KUKA KRL program: MyProgram_018().src

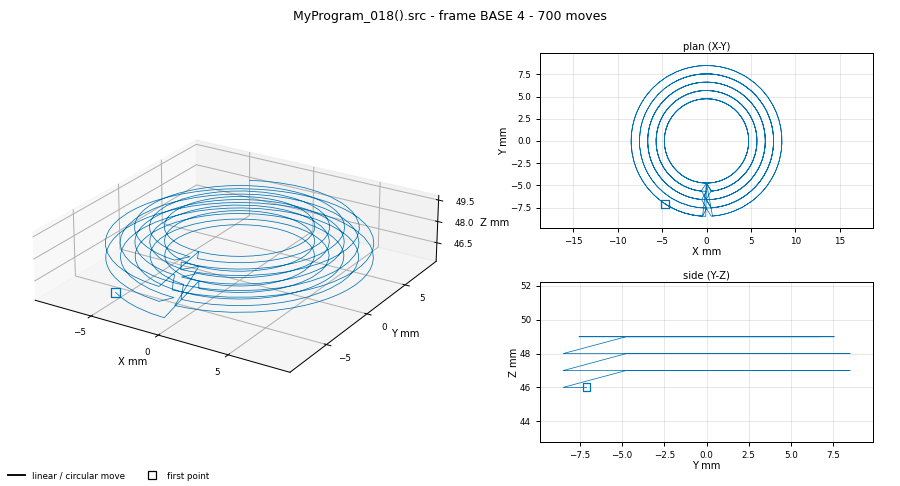
[picture p0: tool path of MyProgram_018().src in frame BASE 4, 700 of 700 moves have a stored position in this frame; points joined in program order, loops and branches not executed]
&ACCESS RVP
&REL 1
&PARAM TEMPLATE = C:\KRC\Roboter\Template\vorgabe
&PARAM EDITMASK = *
DEF MyProgram_018()
; ---- Setting reference (Base) ----
$BASE = BASE_DATA[4]

; --------------------------
; ---- Setting tool (TCP) ----
$TOOL = TOOL_DATA[3]
; --------------------------

$VEL.CP = VEL_APROX_PRINT
Startdeposition()
$VEL.CP = VEL_PRINT
LIN {X -4.657,Y -7.0952,Z 46,A -3.1359,B 0,C 0,E1 0.1598,E2 90.0712} C_DIS
LIN {X -3.9154,Y -7.53,Z 46,A -3.1272,B 0,C 0,E1 0.1598,E2 90.0712} C_DIS
LIN {X -3.1336,Y -7.8876,Z 46,A -3.1138,B 0,C 0,E1 0.1598,E2 90.0713} C_DIS
LIN {X -2.3197,Y -8.1643,Z 46,A -3.0957,B 0,C 0,E1 0.1598,E2 90.0714} C_DIS
LIN {X -1.1138,Y -8.4186,Z 46,A -3.0624,B 0,C 0,E1 0.1598,E2 90.0714} C_DIS
LIN {X -0.0867,Y -8.4896,Z 46,A -3.0278,B 0,C 0,E1 0.1598,E2 90.0715} C_DIS
Enddeposition()
LIN {X 0.0009,Y -4.7549,Z 47,A -2.851,B 0,C 0,E1 0.1598,E2 90.0604} C_DIS
Startdeposition()
$VEL.CP = VEL_PRINT
LIN {X 0.0009,Y -4.7549,Z 47,A -2.8568,B 0,C 0,E1 0.1598,E2 90.0661} C_DIS
LIN {X -0.8332,Y -4.6769,Z 47,A -2.889,B 0,C 0,E1 0.1598,E2 90.071} C_DIS
LIN {X -1.4834,Y -4.5141,Z 47,A -2.9065,B 0,C 0,E1 0.1598,E2 90.0716} C_DIS
LIN {X -2.1038,Y -4.2602,Z 47,A -2.9185,B 0,C 0,E1 0.1598,E2 90.0716} C_DIS
LIN {X -2.6818,Y -3.9209,Z 47,A -2.9253,B 0,C 0,E1 0.1598,E2 90.0716} C_DIS
LIN {X -3.2068,Y -3.5044,Z 47,A -2.9268,B 0,C 0,E1 0.1598,E2 90.0716} C_DIS
LIN {X -3.668,Y -3.0182,Z 47,A -2.9231,B 0,C 0,E1 0.1598,E2 90.0716} C_DIS
LIN {X -4.0561,Y -2.4717,Z 47,A -2.9141,B 0,C 0,E1 0.1598,E2 90.0716} C_DIS
LIN {X -4.3653,Y -1.8772,Z 47,A -2.9002,B 0,C 0,E1 0.1598,E2 90.0716} C_DIS
LIN {X -4.5856,Y -1.244,Z 47,A -2.8814,B 0,C 0,E1 0.1598,E2 90.0716} C_DIS
LIN {X -4.7134,Y -0.5861,Z 47,A -2.8582,B 0,C 0,E1 0.1598,E2 90.0716} C_DIS
LIN {X -4.7503,Y 0.0831,Z 47,A -2.8312,B 0,C 0,E1 0.1598,E2 90.0716} C_DIS
LIN {X -4.6907,Y 0.7507,Z 47,A -2.8007,B 0,C 0,E1 0.1598,E2 90.0716} C_DIS
LIN {X -4.5372,Y 1.4029,Z 47,A -2.7674,B 0,C 0,E1 0.1598,E2 90.0716} C_DIS
LIN {X -4.2974,Y 2.0289,Z 47,A -2.732,B 0,C 0,E1 0.1598,E2 90.0717} C_DIS
LIN {X -3.9689,Y 2.6132,Z 47,A -2.6952,B 0,C 0,E1 0.1598,E2 90.0718} C_DIS
LIN {X -3.5614,Y 3.1455,Z 47,A -2.6576,B 0,C 0,E1 0.1598,E2 90.0718} C_DIS
LIN {X -3.0827,Y 3.6147,Z 47,A -2.6201,B 0,C 0,E1 0.1598,E2 90.072} C_DIS
LIN {X -2.5433,Y 4.0125,Z 47,A -2.5834,B 0,C 0,E1 0.1598,E2 90.072} C_DIS
LIN {X -1.8762,Y 4.3636,Z 47,A -2.5439,B 0,C 0,E1 0.1598,E2 90.0721} C_DIS
LIN {X -1.3241,Y 4.5617,Z 47,A -2.5152,B 0,C 0,E1 0.1598,E2 90.0721} C_DIS
LIN {X -0.6691,Y 4.7028,Z 47,A -2.4851,B 0,C 0,E1 0.1598,E2 90.0722} C_DIS
LIN {X -0.0005,Y 4.7507,Z 47,A -2.4584,B 0,C 0,E1 0.1598,E2 90.0722} C_DIS
LIN {X 0.6681,Y 4.7041,Z 47,A -2.4358,B 0,C 0,E1 0.1598,E2 90.0723} C_DIS
LIN {X 1.3234,Y 4.5632,Z 47,A -2.4176,B 0,C 0,E1 0.1598,E2 90.0723} C_DIS
LIN {X 1.9524,Y 4.3316,Z 47,A -2.4042,B 0,C 0,E1 0.1598,E2 90.0723} C_DIS
LIN {X 2.5429,Y 4.0145,Z 47,A -2.3959,B 0,C 0,E1 0.1598,E2 90.0723} C_DIS
LIN {X 3.0827,Y 3.6169,Z 47,A -2.3929,B 0,C 0,E1 0.1598,E2 90.0723} C_DIS
LIN {X 3.5609,Y 3.147,Z 47,A -2.3953,B 0,C 0,E1 0.1598,E2 90.0723} C_DIS
LIN {X 3.9682,Y 2.6145,Z 47,A -2.4029,B 0,C 0,E1 0.1598,E2 90.0722} C_DIS
LIN {X 4.2968,Y 2.0301,Z 47,A -2.4157,B 0,C 0,E1 0.1598,E2 90.0722} C_DIS
LIN {X 4.5388,Y 1.4049,Z 47,A -2.4334,B 0,C 0,E1 0.1598,E2 90.0721} C_DIS
LIN {X 4.6912,Y 0.7522,Z 47,A -2.4556,B 0,C 0,E1 0.1598,E2 90.0721} C_DIS
LIN {X 4.7506,Y 0.0846,Z 47,A -2.4818,B 0,C 0,E1 0.1598,E2 90.0721} C_DIS
LIN {X 4.7139,Y -0.5846,Z 47,A -2.5117,B 0,C 0,E1 0.1598,E2 90.072} C_DIS
LIN {X 4.5853,Y -1.2422,Z 47,A -2.5445,B 0,C 0,E1 0.1598,E2 90.072} C_DIS
LIN {X 4.3647,Y -1.875,Z 47,A -2.5796,B 0,C 0,E1 0.1598,E2 90.072} C_DIS
LIN {X 4.0578,Y -2.4707,Z 47,A -2.6163,B 0,C 0,E1 0.1598,E2 90.0719} C_DIS
LIN {X 3.6688,Y -3.0165,Z 47,A -2.6539,B 0,C 0,E1 0.1598,E2 90.0719} C_DIS
LIN {X 3.2079,Y -3.5028,Z 47,A -2.6916,B 0,C 0,E1 0.1598,E2 90.0719} C_DIS
LIN {X 2.6838,Y -3.9208,Z 47,A -2.7287,B 0,C 0,E1 0.1598,E2 90.0719} C_DIS
LIN {X 2.1055,Y -4.2599,Z 47,A -2.7644,B 0,C 0,E1 0.1598,E2 90.0719} C_DIS
LIN {X 1.4853,Y -4.5146,Z 47,A -2.798,B 0,C 0,E1 0.1598,E2 90.0719} C_DIS
LIN {X 0.8353,Y -4.6792,Z 47,A -2.8289,B 0,C 0,E1 0.1598,E2 90.0718} C_DIS
LIN {X 0.0009,Y -4.7549,Z 47,A -2.8628,B 0,C 0,E1 0.1598,E2 90.0718} C_DIS
Enddeposition()
LIN {X 0.0009,Y -4.7549,Z 47,A -2.8628,B 0,C 0,E1 0.1598,E2 90.0718} C_DIS
Startdeposition()
$VEL.CP = VEL_PRINT
LIN {X 0.5845,Y -5.6535,Z 47,A -2.8792,B 0,C 0,E1 0.1598,E2 90.0712} C_DIS
LIN {X 1.3635,Y -5.516,Z 47,A -2.8453,B 0,C 0,E1 0.1598,E2 90.0717} C_DIS
LIN {X 2.1164,Y -5.2737,Z 47,A -2.8073,B 0,C 0,E1 0.1598,E2 90.0718} C_DIS
LIN {X 2.8296,Y -4.9313,Z 47,A -2.7665,B 0,C 0,E1 0.1598,E2 90.0718} C_DIS
LIN {X 3.644,Y -4.3696,Z 47,A -2.7126,B 0,C 0,E1 0.1598,E2 90.0718} C_DIS
LIN {X 4.4191,Y -3.5733,Z 47,A -2.65,B 0,C 0,E1 0.1598,E2 90.0717} C_DIS
LIN {X 4.8686,Y -2.9376,Z 47,A -2.6065,B 0,C 0,E1 0.1598,E2 90.0719} C_DIS
LIN {X 5.2236,Y -2.2443,Z 47,A -2.5638,B 0,C 0,E1 0.1598,E2 90.0719} C_DIS
LIN {X 5.4796,Y -1.5089,Z 47,A -2.523,B 0,C 0,E1 0.1598,E2 90.0719} C_DIS
LIN {X 5.6634,Y -0.553,Z 47,A -2.4751,B 0,C 0,E1 0.1598,E2 90.0717} C_DIS
LIN {X 5.6544,Y 0.5908,Z 47,A -2.4265,B 0,C 0,E1 0.1598,E2 90.0716} C_DIS
LIN {X 5.5114,Y 1.3918,Z 47,A -2.398,B 0,C 0,E1 0.1598,E2 90.072} C_DIS
LIN {X 5.256,Y 2.1645,Z 47,A -2.3745,B 0,C 0,E1 0.1598,E2 90.072} C_DIS
LIN {X 4.8941,Y 2.8933,Z 47,A -2.3568,B 0,C 0,E1 0.1598,E2 90.0721} C_DIS
LIN {X 4.4294,Y 3.5613,Z 47,A -2.3455,B 0,C 0,E1 0.1598,E2 90.0721} C_DIS
LIN {X 3.8744,Y 4.156,Z 47,A -2.3406,B 0,C 0,E1 0.1598,E2 90.0722} C_DIS
LIN {X 3.2418,Y 4.6674,Z 47,A -2.3422,B 0,C 0,E1 0.1598,E2 90.0722} C_DIS
LIN {X 2.5416,Y 5.0813,Z 47,A -2.3505,B 0,C 0,E1 0.1598,E2 90.0723} C_DIS
LIN {X 1.7907,Y 5.394,Z 47,A -2.3649,B 0,C 0,E1 0.1598,E2 90.0723} C_DIS
LIN {X 1.0019,Y 5.593,Z 47,A -2.3856,B 0,C 0,E1 0.1598,E2 90.0723} C_DIS
LIN {X 0.1932,Y 5.681,Z 47,A -2.4117,B 0,C 0,E1 0.1598,E2 90.0723} C_DIS
LIN {X -0.6199,Y 5.6502,Z 47,A -2.443,B 0,C 0,E1 0.1598,E2 90.0723} C_DIS
LIN {X -1.4201,Y 5.5034,Z 47,A -2.4787,B 0,C 0,E1 0.1598,E2 90.0723} C_DIS
LIN {X -2.1916,Y 5.245,Z 47,A -2.5181,B 0,C 0,E1 0.1598,E2 90.0722} C_DIS
LIN {X -2.9184,Y 4.8789,Z 47,A -2.5604,B 0,C 0,E1 0.1598,E2 90.0721} C_DIS
LIN {X -3.5851,Y 4.4121,Z 47,A -2.6047,B 0,C 0,E1 0.1598,E2 90.072} C_DIS
LIN {X -4.1768,Y 3.8535,Z 47,A -2.6501,B 0,C 0,E1 0.1598,E2 90.0719} C_DIS
LIN {X -4.6841,Y 3.2176,Z 47,A -2.6957,B 0,C 0,E1 0.1598,E2 90.0718} C_DIS
LIN {X -5.0977,Y 2.5169,Z 47,A -2.7406,B 0,C 0,E1 0.1598,E2 90.0717} C_DIS
LIN {X -5.4038,Y 1.763,Z 47,A -2.7838,B 0,C 0,E1 0.1598,E2 90.0716} C_DIS
LIN {X -5.5993,Y 0.9732,Z 47,A -2.8244,B 0,C 0,E1 0.1598,E2 90.0715} C_DIS
LIN {X -5.6821,Y 0.1638,Z 47,A -2.8617,B 0,C 0,E1 0.1598,E2 90.0715} C_DIS
LIN {X -5.6465,Y -0.649,Z 47,A -2.8949,B 0,C 0,E1 0.1598,E2 90.0714} C_DIS
LIN {X -5.4944,Y -1.4482,Z 47,A -2.9232,B 0,C 0,E1 0.1598,E2 90.0714} C_DIS
LIN {X -5.2319,Y -2.218,Z 47,A -2.9462,B 0,C 0,E1 0.1598,E2 90.0714} C_DIS
LIN {X -4.8611,Y -2.942,Z 47,A -2.9633,B 0,C 0,E1 0.1598,E2 90.0714} C_DIS
LIN {X -4.3918,Y -3.6064,Z 47,A -2.9743,B 0,C 0,E1 0.1598,E2 90.0714} C_DIS
LIN {X -3.8323,Y -4.1971,Z 47,A -2.9789,B 0,C 0,E1 0.1598,E2 90.0714} C_DIS
LIN {X -3.1933,Y -4.7007,Z 47,A -2.9769,B 0,C 0,E1 0.1598,E2 90.0714} C_DIS
LIN {X -2.4901,Y -5.1097,Z 47,A -2.9685,B 0,C 0,E1 0.1598,E2 90.0715} C_DIS
LIN {X -1.4186,Y -5.5098,Z 47,A -2.9462,B 0,C 0,E1 0.1598,E2 90.0715} C_DIS
LIN {X -0.5416,Y -5.6596,Z 47,A -2.9205,B 0,C 0,E1 0.1598,E2 90.0717} C_DIS
LIN {X -0.5416,Y -5.6596,Z 47,A -2.9205,B 0,C 0,E1 0.1598,E2 90.0717} C_DIS
Enddeposition()
LIN {X -0.0004,Y -6.6209,Z 47,A -2.9405,B 0,C 0,E1 0.1598,E2 90.0704} C_DIS
Startdeposition()
$VEL.CP = VEL_PRINT
LIN {X -0.8572,Y -6.5654,Z 47,A -2.9707,B 0,C 0,E1 0.1598,E2 90.0715} C_DIS
LIN {X -1.5328,Y -6.4411,Z 47,A -2.9903,B 0,C 0,E1 0.1598,E2 90.0715} C_DIS
LIN {X -2.1919,Y -6.2476,Z 47,A -3.0062,B 0,C 0,E1 0.1598,E2 90.0715} C_DIS
LIN {X -2.8275,Y -5.9868,Z 47,A -3.0184,B 0,C 0,E1 0.1598,E2 90.0715} C_DIS
LIN {X -3.4329,Y -5.662,Z 47,A -3.0268,B 0,C 0,E1 0.1598,E2 90.0715} C_DIS
LIN {X -4.0011,Y -5.276,Z 47,A -3.0312,B 0,C 0,E1 0.1598,E2 90.0715} C_DIS
LIN {X -4.5248,Y -4.8313,Z 47,A -3.0315,B 0,C 0,E1 0.1598,E2 90.0715} C_DIS
LIN {X -5.0025,Y -4.3375,Z 47,A -3.0281,B 0,C 0,E1 0.1598,E2 90.0715} C_DIS
LIN {X -5.4238,Y -3.7949,Z 47,A -3.0205,B 0,C 0,E1 0.1598,E2 90.0714} C_DIS
LIN {X -5.79,Y -3.2135,Z 47,A -3.0092,B 0,C 0,E1 0.1598,E2 90.0714} C_DIS
LIN {X -6.0918,Y -2.5964,Z 47,A -2.9941,B 0,C 0,E1 0.1598,E2 90.0714} C_DIS
LIN {X -6.328,Y -1.9512,Z 47,A -2.9754,B 0,C 0,E1 0.1598,E2 90.0714} C_DIS
LIN {X -6.4952,Y -1.2848,Z 47,A -2.9533,B 0,C 0,E1 0.1598,E2 90.0714} C_DIS
LIN {X -6.5923,Y -0.6048,Z 47,A -2.928,B 0,C 0,E1 0.1598,E2 90.0714} C_DIS
LIN {X -6.6189,Y 0.0816,Z 47,A -2.8999,B 0,C 0,E1 0.1598,E2 90.0714} C_DIS
LIN {X -6.5767,Y 0.7673,Z 47,A -2.8693,B 0,C 0,E1 0.1598,E2 90.0714} C_DIS
LIN {X -6.4588,Y 1.4441,Z 47,A -2.8363,B 0,C 0,E1 0.1598,E2 90.0715} C_DIS
LIN {X -6.2759,Y 2.1062,Z 47,A -2.8016,B 0,C 0,E1 0.1598,E2 90.0716} C_DIS
LIN {X -6.0234,Y 2.7451,Z 47,A -2.7652,B 0,C 0,E1 0.1598,E2 90.0716} C_DIS
LIN {X -5.7069,Y 3.3548,Z 47,A -2.7278,B 0,C 0,E1 0.1598,E2 90.0717} C_DIS
LIN {X -5.3285,Y 3.9281,Z 47,A -2.6896,B 0,C 0,E1 0.1598,E2 90.0718} C_DIS
LIN {X -4.8934,Y 4.4596,Z 47,A -2.651,B 0,C 0,E1 0.1598,E2 90.0718} C_DIS
LIN {X -4.4045,Y 4.9422,Z 47,A -2.6126,B 0,C 0,E1 0.1598,E2 90.072} C_DIS
LIN {X -3.8687,Y 5.3721,Z 47,A -2.5747,B 0,C 0,E1 0.1598,E2 90.072} C_DIS
LIN {X -3.2907,Y 5.7433,Z 47,A -2.5376,B 0,C 0,E1 0.1598,E2 90.0721} C_DIS
LIN {X -2.3611,Y 6.1883,Z 47,A -2.4845,B 0,C 0,E1 0.1598,E2 90.0721} C_DIS
LIN {X -1.5325,Y 6.4393,Z 47,A -2.4433,B 0,C 0,E1 0.1598,E2 90.0723} C_DIS
LIN {X -0.8516,Y 6.5656,Z 47,A -2.4129,B 0,C 0,E1 0.1598,E2 90.0723} C_DIS
LIN {X -0.1612,Y 6.6195,Z 47,A -2.3851,B 0,C 0,E1 0.1598,E2 90.0723} C_DIS
LIN {X 0.5311,Y 6.5989,Z 47,A -2.3605,B 0,C 0,E1 0.1598,E2 90.0724} C_DIS
LIN {X 1.2176,Y 6.508,Z 47,A -2.339,B 0,C 0,E1 0.1598,E2 90.0724} C_DIS
LIN {X 1.8908,Y 6.3452,Z 47,A -2.3211,B 0,C 0,E1 0.1598,E2 90.0724} C_DIS
LIN {X 2.5429,Y 6.1122,Z 47,A -2.3069,B 0,C 0,E1 0.1598,E2 90.0724} C_DIS
LIN {X 3.1673,Y 5.8123,Z 47,A -2.2966,B 0,C 0,E1 0.1598,E2 90.0724} C_DIS
LIN {X 3.7569,Y 5.4491,Z 47,A -2.2903,B 0,C 0,E1 0.1598,E2 90.0724} C_DIS
LIN {X 4.3059,Y 5.0269,Z 47,A -2.288,B 0,C 0,E1 0.1598,E2 90.0724} C_DIS
LIN {X 4.8068,Y 4.5488,Z 47,A -2.2898,B 0,C 0,E1 0.1598,E2 90.0724} C_DIS
LIN {X 5.2576,Y 4.0231,Z 47,A -2.2956,B 0,C 0,E1 0.1598,E2 90.0724} C_DIS
LIN {X 5.6506,Y 3.4527,Z 47,A -2.3054,B 0,C 0,E1 0.1598,E2 90.0723} C_DIS
LIN {X 5.9786,Y 2.8428,Z 47,A -2.3193,B 0,C 0,E1 0.1598,E2 90.0723} C_DIS
LIN {X 6.2421,Y 2.2022,Z 47,A -2.3369,B 0,C 0,E1 0.1598,E2 90.0723} C_DIS
LIN {X 6.4381,Y 1.538,Z 47,A -2.358,B 0,C 0,E1 0.1598,E2 90.0722} C_DIS
LIN {X 6.565,Y 0.8572,Z 47,A -2.3823,B 0,C 0,E1 0.1598,E2 90.0722} C_DIS
LIN {X 6.6166,Y 0.1667,Z 47,A -2.4099,B 0,C 0,E1 0.1598,E2 90.0721} C_DIS
LIN {X 6.5989,Y -0.5256,Z 47,A -2.4401,B 0,C 0,E1 0.1598,E2 90.0721} C_DIS
LIN {X 6.5074,Y -1.212,Z 47,A -2.4727,B 0,C 0,E1 0.1598,E2 90.0721} C_DIS
LIN {X 6.3463,Y -1.8856,Z 47,A -2.5074,B 0,C 0,E1 0.1598,E2 90.072} C_DIS
LIN {X 6.1156,Y -2.5387,Z 47,A -2.5438,B 0,C 0,E1 0.1598,E2 90.072} C_DIS
LIN {X 5.8167,Y -3.1636,Z 47,A -2.5815,B 0,C 0,E1 0.1598,E2 90.072} C_DIS
LIN {X 5.454,Y -3.7537,Z 47,A -2.62,B 0,C 0,E1 0.1598,E2 90.0719} C_DIS
LIN {X 5.0333,Y -4.3041,Z 47,A -2.659,B 0,C 0,E1 0.1598,E2 90.0719} C_DIS
LIN {X 4.5562,Y -4.8062,Z 47,A -2.6979,B 0,C 0,E1 0.1598,E2 90.0719} C_DIS
LIN {X 4.0291,Y -5.2557,Z 47,A -2.7365,B 0,C 0,E1 0.1598,E2 90.0719} C_DIS
LIN {X 3.4569,Y -5.646,Z 47,A -2.7742,B 0,C 0,E1 0.1598,E2 90.0719} C_DIS
LIN {X 2.8484,Y -5.9768,Z 47,A -2.8106,B 0,C 0,E1 0.1598,E2 90.0718} C_DIS
LIN {X 2.2087,Y -6.242,Z 47,A -2.8454,B 0,C 0,E1 0.1598,E2 90.0718} C_DIS
LIN {X 1.5443,Y -6.4372,Z 47,A -2.8781,B 0,C 0,E1 0.1598,E2 90.0718} C_DIS
LIN {X 0.8632,Y -6.5628,Z 47,A -2.9085,B 0,C 0,E1 0.1598,E2 90.0717} C_DIS
LIN {X -0.0004,Y -6.6209,Z 47,A -2.9426,B 0,C 0,E1 0.1598,E2 90.0717} C_DIS
Enddeposition()
LIN {X -0.0004,Y -6.6209,Z 47,A -2.9426,B 0,C 0,E1 0.1598,E2 90.0717} C_DIS
Startdeposition()
$VEL.CP = VEL_PRINT
LIN {X 0.5272,Y -7.5354,Z 47,A -2.9618,B 0,C 0,E1 0.1598,E2 90.071} C_DIS
LIN {X 1.3696,Y -7.4334,Z 47,A -2.9271,B 0,C 0,E1 0.1598,E2 90.0716} C_DIS
LIN {X 2.5106,Y -7.1281,Z 47,A -2.8723,B 0,C 0,E1 0.1598,E2 90.0716} C_DIS
LIN {X 3.5797,Y -6.6516,Z 47,A -2.8127,B 0,C 0,E1 0.1598,E2 90.0716} C_DIS
LIN {X 4.2345,Y -6.2589,Z 47,A -2.7719,B 0,C 0,E1 0.1598,E2 90.0718} C_DIS
LIN {X 4.9755,Y -5.6846,Z 47,A -2.7202,B 0,C 0,E1 0.1598,E2 90.0718} C_DIS
LIN {X 5.5133,Y -5.162,Z 47,A -2.6781,B 0,C 0,E1 0.1598,E2 90.0718} C_DIS
LIN {X 5.9992,Y -4.5907,Z 47,A -2.6359,B 0,C 0,E1 0.1598,E2 90.0718} C_DIS
LIN {X 6.4246,Y -3.9733,Z 47,A -2.5938,B 0,C 0,E1 0.1598,E2 90.0719} C_DIS
LIN {X 6.8711,Y -3.149,Z 47,A -2.542,B 0,C 0,E1 0.1598,E2 90.0718} C_DIS
LIN {X 7.2591,Y -2.0861,Z 47,A -2.4821,B 0,C 0,E1 0.1598,E2 90.0716} C_DIS
LIN {X 7.4329,Y -1.346,Z 47,A -2.4444,B 0,C 0,E1 0.1598,E2 90.072} C_DIS
LIN {X 7.5535,Y -0.2415,Z 47,A -2.3925,B 0,C 0,E1 0.1598,E2 90.0717} C_DIS
LIN {X 7.521,Y 0.6923,Z 47,A -2.354,B 0,C 0,E1 0.1598,E2 90.072} C_DIS
LIN {X 7.4162,Y 1.4323,Z 47,A -2.3264,B 0,C 0,E1 0.1598,E2 90.0721} C_DIS
LIN {X 7.239,Y 2.1584,Z 47,A -2.302,B 0,C 0,E1 0.1598,E2 90.0721} C_DIS
LIN {X 6.8418,Y 3.2096,Z 47,A -2.2714,B 0,C 0,E1 0.1598,E2 90.0719} C_DIS
LIN {X 6.4285,Y 3.9665,Z 47,A -2.2547,B 0,C 0,E1 0.1598,E2 90.0722} C_DIS
LIN {X 5.785,Y 4.8618,Z 47,A -2.2401,B 0,C 0,E1 0.1598,E2 90.0721} C_DIS
LIN {X 5.0845,Y 5.5857,Z 47,A -2.2352,B 0,C 0,E1 0.1598,E2 90.0723} C_DIS
LIN {X 4.4605,Y 6.0956,Z 47,A -2.2367,B 0,C 0,E1 0.1598,E2 90.0724} C_DIS
LIN {X 3.6114,Y 6.6377,Z 47,A -2.2449,B 0,C 0,E1 0.1598,E2 90.0724} C_DIS
LIN {X 2.5888,Y 7.0993,Z 47,A -2.263,B 0,C 0,E1 0.1598,E2 90.0724} C_DIS
LIN {X 1.3636,Y 7.4345,Z 47,A -2.2941,B 0,C 0,E1 0.1598,E2 90.0724} C_DIS
LIN {X 0.4621,Y 7.5429,Z 47,A -2.3228,B 0,C 0,E1 0.1598,E2 90.0724} C_DIS
LIN {X -0.6975,Y 7.5262,Z 47,A -2.3663,B 0,C 0,E1 0.1598,E2 90.0724} C_DIS
LIN {X -1.5379,Y 7.3986,Z 47,A -2.4028,B 0,C 0,E1 0.1598,E2 90.0724} C_DIS
LIN {X -2.6885,Y 7.0592,Z 47,A -2.4595,B 0,C 0,E1 0.1598,E2 90.0722} C_DIS
LIN {X -3.8311,Y 6.5146,Z 47,A -2.5247,B 0,C 0,E1 0.1598,E2 90.0721} C_DIS
LIN {X -4.6142,Y 5.984,Z 47,A -2.576,B 0,C 0,E1 0.1598,E2 90.072} C_DIS
LIN {X -5.4462,Y 5.2327,Z 47,A -2.6384,B 0,C 0,E1 0.1598,E2 90.0718} C_DIS
LIN {X -6.0843,Y 4.4839,Z 47,A -2.6935,B 0,C 0,E1 0.1598,E2 90.0716} C_DIS
LIN {X -6.6875,Y 3.5096,Z 47,A -2.7568,B 0,C 0,E1 0.1598,E2 90.0714} C_DIS
LIN {X -7.1184,Y 2.537,Z 47,A -2.8138,B 0,C 0,E1 0.1598,E2 90.0712} C_DIS
LIN {X -7.4177,Y 1.4469,Z 47,A -2.8709,B 0,C 0,E1 0.1598,E2 90.0712} C_DIS
LIN {X -7.5503,Y 0.2333,Z 47,A -2.9269,B 0,C 0,E1 0.1598,E2 90.0708} C_DIS
LIN {X -7.5352,Y -0.5765,Z 47,A -2.961,B 0,C 0,E1 0.1598,E2 90.0711} C_DIS
LIN {X -7.3683,Y -1.6658,Z 47,A -3.0008,B 0,C 0,E1 0.1598,E2 90.0709} C_DIS
LIN {X -7.1524,Y -2.4273,Z 47,A -3.0255,B 0,C 0,E1 0.1598,E2 90.0712} C_DIS
LIN {X -6.8586,Y -3.1621,Z 47,A -3.0459,B 0,C 0,E1 0.1598,E2 90.0712} C_DIS
LIN {X -6.4896,Y -3.8623,Z 47,A -3.062,B 0,C 0,E1 0.1598,E2 90.0712} C_DIS
LIN {X -6.0495,Y -4.5199,Z 47,A -3.0738,B 0,C 0,E1 0.1598,E2 90.0712} C_DIS
LIN {X -5.5432,Y -5.1281,Z 47,A -3.0811,B 0,C 0,E1 0.1598,E2 90.0712} C_DIS
LIN {X -4.9766,Y -5.6805,Z 47,A -3.0838,B 0,C 0,E1 0.1598,E2 90.0712} C_DIS
LIN {X -4.0505,Y -6.3798,Z 47,A -3.0794,B 0,C 0,E1 0.1598,E2 90.0712} C_DIS
LIN {X -3.0631,Y -6.903,Z 47,A -3.0655,B 0,C 0,E1 0.1598,E2 90.0713} C_DIS
LIN {X -1.9291,Y -7.3063,Z 47,A -3.0412,B 0,C 0,E1 0.1598,E2 90.0714} C_DIS
LIN {X -0.8836,Y -7.5051,Z 47,A -3.0114,B 0,C 0,E1 0.1598,E2 90.0715} C_DIS
LIN {X 0.0185,Y -7.5578,Z 47,A -2.9806,B 0,C 0,E1 0.1598,E2 90.0715} C_DIS
Enddeposition()
LIN {X 0.0185,Y -7.5578,Z 47,A -2.9806,B 0,C 0,E1 0.1598,E2 90.0715} C_DIS
Startdeposition()
$VEL.CP = VEL_PRINT
LIN {X -0.4519,Y -8.4793,Z 47,A -3.0367,B 0,C 0,E1 0.1598,E2 90.0709} C_DIS
LIN {X -1.6061,Y -8.3325,Z 47,A -3.0733,B 0,C 0,E1 0.1598,E2 90.0714} C_DIS
LIN {X -2.4329,Y -8.1295,Z 47,A -3.0949,B 0,C 0,E1 0.1598,E2 90.0714} C_DIS
LIN {X -3.2351,Y -7.8449,Z 47,A -3.1122,B 0,C 0,E1 0.1598,E2 90.0714} C_DIS
LIN {X -4.0049,Y -7.4813,Z 47,A -3.1249,B 0,C 0,E1 0.1598,E2 90.0714} C_DIS
LIN {X -4.7343,Y -7.0424,Z 47,A -3.133,B 0,C 0,E1 0.1598,E2 90.0713} C_DIS
LIN {X -5.4161,Y -6.5327,Z 47,A -3.1363,B 0,C 0,E1 0.1598,E2 90.0713} C_DIS
LIN {X -6.0435,Y -5.9572,Z 47,A -3.1349,B 0,C 0,E1 0.1598,E2 90.0713} C_DIS
LIN {X -6.6102,Y -5.3219,Z 47,A -3.1287,B 0,C 0,E1 0.1598,E2 90.0712} C_DIS
LIN {X -7.1104,Y -4.633,Z 47,A -3.1178,B 0,C 0,E1 0.1598,E2 90.0712} C_DIS
LIN {X -7.5391,Y -3.8974,Z 47,A -3.1023,B 0,C 0,E1 0.1598,E2 90.0712} C_DIS
LIN {X -7.8918,Y -3.1225,Z 47,A -3.0824,B 0,C 0,E1 0.1598,E2 90.0712} C_DIS
LIN {X -8.1652,Y -2.3162,Z 47,A -3.0582,B 0,C 0,E1 0.1598,E2 90.0712} C_DIS
LIN {X -8.3566,Y -1.4865,Z 47,A -3.0301,B 0,C 0,E1 0.1598,E2 90.0712} C_DIS
LIN {X -8.4851,Y -0.3389,Z 47,A -2.986,B 0,C 0,E1 0.1598,E2 90.0709} C_DIS
LIN {X -8.4649,Y 0.6668,Z 47,A -2.9427,B 0,C 0,E1 0.1598,E2 90.0711} C_DIS
LIN {X -8.3114,Y 1.7339,Z 47,A -2.8919,B 0,C 0,E1 0.1598,E2 90.0711} C_DIS
LIN {X -8.0194,Y 2.7788,Z 47,A -2.837,B 0,C 0,E1 0.1598,E2 90.0713} C_DIS
LIN {X -7.5555,Y 3.8768,Z 47,A -2.7734,B 0,C 0,E1 0.1598,E2 90.0713} C_DIS
LIN {X -6.9083,Y 4.9371,Z 47,A -2.7046,B 0,C 0,E1 0.1598,E2 90.0713} C_DIS
LIN {X -6.2032,Y 5.797,Z 47,A -2.6425,B 0,C 0,E1 0.1598,E2 90.0716} C_DIS
LIN {X -5.4008,Y 6.5471,Z 47,A -2.5813,B 0,C 0,E1 0.1598,E2 90.0719} C_DIS
LIN {X -4.5118,Y 7.1922,Z 47,A -2.5212,B 0,C 0,E1 0.1598,E2 90.0719} C_DIS
LIN {X -3.3607,Y 7.7968,Z 47,A -2.4531,B 0,C 0,E1 0.1598,E2 90.0721} C_DIS
LIN {X -2.103,Y 8.2258,Z 47,A -2.3886,B 0,C 0,E1 0.1598,E2 90.0723} C_DIS
LIN {X -0.9642,Y 8.4337,Z 47,A -2.3378,B 0,C 0,E1 0.1598,E2 90.0724} C_DIS
LIN {X -0.126,Y 8.4871,Z 47,A -2.3046,B 0,C 0,E1 0.1598,E2 90.0724} C_DIS
LIN {X 0.7132,Y 8.4571,Z 47,A -2.2749,B 0,C 0,E1 0.1598,E2 90.0725} C_DIS
LIN {X 1.5454,Y 8.3445,Z 47,A -2.249,B 0,C 0,E1 0.1598,E2 90.0725} C_DIS
LIN {X 2.3627,Y 8.1511,Z 47,A -2.227,B 0,C 0,E1 0.1598,E2 90.0725} C_DIS
LIN {X 3.157,Y 7.8781,Z 47,A -2.2093,B 0,C 0,E1 0.1598,E2 90.0725} C_DIS
LIN {X 4.314,Y 7.3145,Z 47,A -2.1904,B 0,C 0,E1 0.1598,E2 90.0725} C_DIS
LIN {X 5.4016,Y 6.5457,Z 47,A -2.1828,B 0,C 0,E1 0.1598,E2 90.0723} C_DIS
LIN {X 6.3218,Y 5.6702,Z 47,A -2.1861,B 0,C 0,E1 0.1598,E2 90.0722} C_DIS
LIN {X 6.9271,Y 4.9098,Z 47,A -2.1962,B 0,C 0,E1 0.1598,E2 90.0722} C_DIS
LIN {X 7.4924,Y 3.9877,Z 47,A -2.2146,B 0,C 0,E1 0.1598,E2 90.0722} C_DIS
LIN {X 7.8592,Y 3.204,Z 47,A -2.2346,B 0,C 0,E1 0.1598,E2 90.0722} C_DIS
LIN {X 8.1443,Y 2.3871,Z 47,A -2.259,B 0,C 0,E1 0.1598,E2 90.0722} C_DIS
LIN {X 8.3451,Y 1.5455,Z 47,A -2.2875,B 0,C 0,E1 0.1598,E2 90.0721} C_DIS
LIN {X 8.4591,Y 0.6878,Z 47,A -2.3199,B 0,C 0,E1 0.1598,E2 90.0721} C_DIS
LIN {X 8.4861,Y -0.1769,Z 47,A -2.3559,B 0,C 0,E1 0.1598,E2 90.072} C_DIS
LIN {X 8.4228,Y -1.0398,Z 47,A -2.3951,B 0,C 0,E1 0.1598,E2 90.072} C_DIS
LIN {X 8.273,Y -1.8919,Z 47,A -2.437,B 0,C 0,E1 0.1598,E2 90.072} C_DIS
LIN {X 8.0375,Y -2.7245,Z 47,A -2.4812,B 0,C 0,E1 0.1598,E2 90.0719} C_DIS
LIN {X 7.7185,Y -3.5287,Z 47,A -2.5274,B 0,C 0,E1 0.1598,E2 90.0719} C_DIS
LIN {X 7.3192,Y -4.2963,Z 47,A -2.5749,B 0,C 0,E1 0.1598,E2 90.0719} C_DIS
LIN {X 6.8438,Y -5.0193,Z 47,A -2.6232,B 0,C 0,E1 0.1598,E2 90.0718} C_DIS
LIN {X 6.1521,Y -5.8508,Z 47,A -2.684,B 0,C 0,E1 0.1598,E2 90.0716} C_DIS
LIN {X 5.2427,Y -6.6784,Z 47,A -2.7528,B 0,C 0,E1 0.1598,E2 90.0716} C_DIS
LIN {X 4.0942,Y -7.4377,Z 47,A -2.8274,B 0,C 0,E1 0.1598,E2 90.0716} C_DIS
LIN {X 3.1368,Y -7.8853,Z 47,A -2.8817,B 0,C 0,E1 0.1598,E2 90.0716} C_DIS
LIN {X 2.3367,Y -8.1586,Z 47,A -2.9228,B 0,C 0,E1 0.1598,E2 90.0716} C_DIS
LIN {X 1.5133,Y -8.3512,Z 47,A -2.9612,B 0,C 0,E1 0.1598,E2 90.0716} C_DIS
LIN {X 0.6748,Y -8.461,Z 47,A -2.9966,B 0,C 0,E1 0.1598,E2 90.0716} C_DIS
LIN {X 0.6748,Y -8.461,Z 47,A -2.9966,B 0,C 0,E1 0.1598,E2 90.0716} C_DIS
Enddeposition()
LIN {X 0.0009,Y -4.7523,Z 48,A -2.8488,B 0,C 0,E1 0.1598,E2 90.0604} C_DIS
Startdeposition()
$VEL.CP = VEL_PRINT
LIN {X 0.0009,Y -4.7523,Z 48,A -2.8545,B 0,C 0,E1 0.1598,E2 90.0661} C_DIS
LIN {X 0.8354,Y -4.679,Z 48,A -2.8257,B 0,C 0,E1 0.1598,E2 90.0711} C_DIS
LIN {X 1.4853,Y -4.5141,Z 48,A -2.7955,B 0,C 0,E1 0.1598,E2 90.0718} C_DIS
LIN {X 2.1051,Y -4.2586,Z 48,A -2.7619,B 0,C 0,E1 0.1598,E2 90.0718} C_DIS
LIN {X 2.6838,Y -3.9204,Z 48,A -2.7262,B 0,C 0,E1 0.1598,E2 90.0718} C_DIS
LIN {X 3.2088,Y -3.5037,Z 48,A -2.6891,B 0,C 0,E1 0.1598,E2 90.0718} C_DIS
LIN {X 3.6692,Y -3.0166,Z 48,A -2.6514,B 0,C 0,E1 0.1598,E2 90.0719} C_DIS
LIN {X 4.0591,Y -2.4714,Z 48,A -2.6138,B 0,C 0,E1 0.1598,E2 90.0719} C_DIS
LIN {X 4.3643,Y -1.8744,Z 48,A -2.5771,B 0,C 0,E1 0.1598,E2 90.0719} C_DIS
LIN {X 4.5854,Y -1.2419,Z 48,A -2.5419,B 0,C 0,E1 0.1598,E2 90.0719} C_DIS
LIN {X 4.7142,Y -0.5843,Z 48,A -2.5091,B 0,C 0,E1 0.1598,E2 90.0719} C_DIS
LIN {X 4.7506,Y 0.0849,Z 48,A -2.4792,B 0,C 0,E1 0.1598,E2 90.072} C_DIS
LIN {X 4.6911,Y 0.7526,Z 48,A -2.4529,B 0,C 0,E1 0.1598,E2 90.072} C_DIS
LIN {X 4.5389,Y 1.4053,Z 48,A -2.4307,B 0,C 0,E1 0.1598,E2 90.072} C_DIS
LIN {X 4.2967,Y 2.0305,Z 48,A -2.413,B 0,C 0,E1 0.1598,E2 90.0721} C_DIS
LIN {X 3.9681,Y 2.6148,Z 48,A -2.4002,B 0,C 0,E1 0.1598,E2 90.0721} C_DIS
LIN {X 3.5608,Y 3.1474,Z 48,A -2.3926,B 0,C 0,E1 0.1598,E2 90.0722} C_DIS
LIN {X 3.0824,Y 3.6171,Z 48,A -2.3903,B 0,C 0,E1 0.1598,E2 90.0722} C_DIS
LIN {X 2.5424,Y 4.0145,Z 48,A -2.3933,B 0,C 0,E1 0.1598,E2 90.0722} C_DIS
LIN {X 1.952,Y 4.3317,Z 48,A -2.4016,B 0,C 0,E1 0.1598,E2 90.0723} C_DIS
LIN {X 1.323,Y 4.5633,Z 48,A -2.4149,B 0,C 0,E1 0.1598,E2 90.0723} C_DIS
LIN {X 0.6677,Y 4.7041,Z 48,A -2.4331,B 0,C 0,E1 0.1598,E2 90.0723} C_DIS
LIN {X -0.001,Y 4.7507,Z 48,A -2.4558,B 0,C 0,E1 0.1598,E2 90.0723} C_DIS
LIN {X -0.6694,Y 4.7026,Z 48,A -2.4825,B 0,C 0,E1 0.1598,E2 90.0723} C_DIS
LIN {X -1.3247,Y 4.5622,Z 48,A -2.5126,B 0,C 0,E1 0.1598,E2 90.0723} C_DIS
LIN {X -1.9538,Y 4.331,Z 48,A -2.5456,B 0,C 0,E1 0.1598,E2 90.0722} C_DIS
LIN {X -2.5436,Y 4.0126,Z 48,A -2.5808,B 0,C 0,E1 0.1598,E2 90.0721} C_DIS
LIN {X -3.0832,Y 3.615,Z 48,A -2.6175,B 0,C 0,E1 0.1598,E2 90.0721} C_DIS
LIN {X -3.5614,Y 3.1453,Z 48,A -2.655,B 0,C 0,E1 0.1598,E2 90.0719} C_DIS
LIN {X -3.9692,Y 2.6132,Z 48,A -2.6926,B 0,C 0,E1 0.1598,E2 90.0719} C_DIS
LIN {X -4.298,Y 2.0289,Z 48,A -2.7294,B 0,C 0,E1 0.1598,E2 90.0718} C_DIS
LIN {X -4.5409,Y 1.404,Z 48,A -2.7648,B 0,C 0,E1 0.1598,E2 90.0717} C_DIS
LIN {X -4.6929,Y 0.751,Z 48,A -2.7981,B 0,C 0,E1 0.1598,E2 90.0717} C_DIS
LIN {X -4.752,Y 0.0831,Z 48,A -2.8286,B 0,C 0,E1 0.1598,E2 90.0716} C_DIS
LIN {X -4.7151,Y -0.5862,Z 48,A -2.8556,B 0,C 0,E1 0.1598,E2 90.0716} C_DIS
LIN {X -4.5853,Y -1.2437,Z 48,A -2.8787,B 0,C 0,E1 0.1598,E2 90.0716} C_DIS
LIN {X -4.3648,Y -1.8768,Z 48,A -2.8975,B 0,C 0,E1 0.1598,E2 90.0715} C_DIS
LIN {X -4.0561,Y -2.4717,Z 48,A -2.9114,B 0,C 0,E1 0.1598,E2 90.0715} C_DIS
LIN {X -3.6681,Y -3.0181,Z 48,A -2.9204,B 0,C 0,E1 0.1598,E2 90.0715} C_DIS
LIN {X -3.2069,Y -3.5044,Z 48,A -2.9242,B 0,C 0,E1 0.1598,E2 90.0715} C_DIS
LIN {X -2.6818,Y -3.9209,Z 48,A -2.9226,B 0,C 0,E1 0.1598,E2 90.0715} C_DIS
LIN {X -2.1038,Y -4.2601,Z 48,A -2.9158,B 0,C 0,E1 0.1598,E2 90.0716} C_DIS
LIN {X -1.4834,Y -4.5139,Z 48,A -2.9039,B 0,C 0,E1 0.1598,E2 90.0716} C_DIS
LIN {X -0.8332,Y -4.6765,Z 48,A -2.887,B 0,C 0,E1 0.1598,E2 90.0717} C_DIS
LIN {X 0.0009,Y -4.7523,Z 48,A -2.8596,B 0,C 0,E1 0.1598,E2 90.0717} C_DIS
Enddeposition()
LIN {X 0.0009,Y -4.7523,Z 48,A -2.8596,B 0,C 0,E1 0.1598,E2 90.0717} C_DIS
Startdeposition()
$VEL.CP = VEL_PRINT
LIN {X -0.619,Y -5.651,Z 48,A -2.9201,B 0,C 0,E1 0.1598,E2 90.0711} C_DIS
LIN {X -1.3975,Y -5.5101,Z 48,A -2.9432,B 0,C 0,E1 0.1598,E2 90.0716} C_DIS
LIN {X -2.1483,Y -5.2609,Z 48,A -2.9602,B 0,C 0,E1 0.1598,E2 90.0716} C_DIS
LIN {X -2.8588,Y -4.9133,Z 48,A -2.9715,B 0,C 0,E1 0.1598,E2 90.0716} C_DIS
LIN {X -3.5132,Y -4.4689,Z 48,A -2.9765,B 0,C 0,E1 0.1598,E2 90.0715} C_DIS
LIN {X -4.0994,Y -3.9375,Z 48,A -2.9754,B 0,C 0,E1 0.1598,E2 90.0715} C_DIS
LIN {X -4.6072,Y -3.3307,Z 48,A -2.9683,B 0,C 0,E1 0.1598,E2 90.0715} C_DIS
LIN {X -5.0235,Y -2.6581,Z 48,A -2.955,B 0,C 0,E1 0.1598,E2 90.0714} C_DIS
LIN {X -5.3441,Y -1.935,Z 48,A -2.936,B 0,C 0,E1 0.1598,E2 90.0714} C_DIS
LIN {X -5.5592,Y -1.1739,Z 48,A -2.9116,B 0,C 0,E1 0.1598,E2 90.0714} C_DIS
LIN {X -5.6699,Y -0.3909,Z 48,A -2.8825,B 0,C 0,E1 0.1598,E2 90.0714} C_DIS
LIN {X -5.6083,Y 0.96,Z 48,A -2.8222,B 0,C 0,E1 0.1598,E2 90.0708} C_DIS
LIN {X -5.2185,Y 2.2524,Z 48,A -2.7533,B 0,C 0,E1 0.1598,E2 90.0711} C_DIS
LIN {X -4.8375,Y 2.983,Z 48,A -2.7088,B 0,C 0,E1 0.1598,E2 90.0716} C_DIS
LIN {X -4.3552,Y 3.6512,Z 48,A -2.6628,B 0,C 0,E1 0.1598,E2 90.0718} C_DIS
LIN {X -3.7821,Y 4.2434,Z 48,A -2.6166,B 0,C 0,E1 0.1598,E2 90.0719} C_DIS
LIN {X -3.3022,Y 4.6335,Z 48,A -2.5825,B 0,C 0,E1 0.1598,E2 90.0721} C_DIS
LIN {X -2.1046,Y 5.2855,Z 48,A -2.5106,B 0,C 0,E1 0.1598,E2 90.0721} C_DIS
LIN {X -1.0086,Y 5.6005,Z 48,A -2.457,B 0,C 0,E1 0.1598,E2 90.0722} C_DIS
LIN {X -0.0045,Y 5.6906,Z 48,A -2.4162,B 0,C 0,E1 0.1598,E2 90.0723} C_DIS
LIN {X 1.0286,Y 5.5883,Z 48,A -2.3824,B 0,C 0,E1 0.1598,E2 90.0723} C_DIS
LIN {X 1.832,Y 5.3787,Z 48,A -2.3617,B 0,C 0,E1 0.1598,E2 90.0723} C_DIS
LIN {X 2.5963,Y 5.0541,Z 48,A -2.3472,B 0,C 0,E1 0.1598,E2 90.0723} C_DIS
LIN {X 3.3058,Y 4.6226,Z 48,A -2.3394,B 0,C 0,E1 0.1598,E2 90.0723} C_DIS
LIN {X 3.9434,Y 4.0908,Z 48,A -2.3385,B 0,C 0,E1 0.1598,E2 90.0723} C_DIS
LIN {X 4.4975,Y 3.4725,Z 48,A -2.3443,B 0,C 0,E1 0.1598,E2 90.0723} C_DIS
LIN {X 4.9567,Y 2.7807,Z 48,A -2.3569,B 0,C 0,E1 0.1598,E2 90.0721} C_DIS
LIN {X 5.31,Y 2.029,Z 48,A -2.3758,B 0,C 0,E1 0.1598,E2 90.0721} C_DIS
LIN {X 5.549,Y 1.2335,Z 48,A -2.4009,B 0,C 0,E1 0.1598,E2 90.072} C_DIS
LIN {X 5.6704,Y 0.4118,Z 48,A -2.4315,B 0,C 0,E1 0.1598,E2 90.072} C_DIS
LIN {X 5.6693,Y -0.4189,Z 48,A -2.4669,B 0,C 0,E1 0.1598,E2 90.0719} C_DIS
LIN {X 5.5474,Y -1.2405,Z 48,A -2.5065,B 0,C 0,E1 0.1598,E2 90.0719} C_DIS
LIN {X 5.1718,Y -2.3741,Z 48,A -2.5684,B 0,C 0,E1 0.1598,E2 90.0715} C_DIS
LIN {X 4.7244,Y -3.1591,Z 48,A -2.6186,B 0,C 0,E1 0.1598,E2 90.0718} C_DIS
LIN {X 4.286,Y -3.7338,Z 48,A -2.6594,B 0,C 0,E1 0.1598,E2 90.0718} C_DIS
LIN {X 3.7775,Y -4.2472,Z 48,A -2.7,B 0,C 0,E1 0.1598,E2 90.0718} C_DIS
LIN {X 3.2082,Y -4.6928,Z 48,A -2.74,B 0,C 0,E1 0.1598,E2 90.0718} C_DIS
LIN {X 2.5862,Y -5.0609,Z 48,A -2.7785,B 0,C 0,E1 0.1598,E2 90.0718} C_DIS
LIN {X 1.9235,Y -5.3494,Z 48,A -2.8152,B 0,C 0,E1 0.1598,E2 90.0718} C_DIS
LIN {X 1.2297,Y -5.5517,Z 48,A -2.8493,B 0,C 0,E1 0.1598,E2 90.0718} C_DIS
LIN {X 0.5154,Y -5.6625,Z 48,A -2.8802,B 0,C 0,E1 0.1598,E2 90.0718} C_DIS
LIN {X 0.5154,Y -5.6625,Z 48,A -2.8802,B 0,C 0,E1 0.1598,E2 90.0718} C_DIS
Enddeposition()
LIN {X -0.0418,Y -6.6226,Z 48,A -2.9405,B 0,C 0,E1 0.1598,E2 90.0705} C_DIS
Startdeposition()
$VEL.CP = VEL_PRINT
LIN {X 0.8086,Y -6.5706,Z 48,A -2.9082,B 0,C 0,E1 0.1598,E2 90.0716} C_DIS
LIN {X 1.4801,Y -6.4533,Z 48,A -2.8786,B 0,C 0,E1 0.1598,E2 90.0717} C_DIS
LIN {X 2.1353,Y -6.2657,Z 48,A -2.8466,B 0,C 0,E1 0.1598,E2 90.0717} C_DIS
LIN {X 2.7682,Y -6.0127,Z 48,A -2.8126,B 0,C 0,E1 0.1598,E2 90.0717} C_DIS
LIN {X 3.3718,Y -5.6961,Z 48,A -2.7769,B 0,C 0,E1 0.1598,E2 90.0718} C_DIS
LIN {X 3.9402,Y -5.3198,Z 48,A -2.74,B 0,C 0,E1 0.1598,E2 90.0718} C_DIS
LIN {X 4.4653,Y -4.8853,Z 48,A -2.7021,B 0,C 0,E1 0.1598,E2 90.0718} C_DIS
LIN {X 4.9448,Y -4.4009,Z 48,A -2.6638,B 0,C 0,E1 0.1598,E2 90.0718} C_DIS
LIN {X 5.3711,Y -3.8692,Z 48,A -2.6255,B 0,C 0,E1 0.1598,E2 90.0719} C_DIS
LIN {X 5.7406,Y -3.2965,Z 48,A -2.5874,B 0,C 0,E1 0.1598,E2 90.0719} C_DIS
LIN {X 6.0482,Y -2.6883,Z 48,A -2.5501,B 0,C 0,E1 0.1598,E2 90.0719} C_DIS
LIN {X 6.2929,Y -2.0522,Z 48,A -2.514,B 0,C 0,E1 0.1598,E2 90.0719} C_DIS
LIN {X 6.4699,Y -1.3941,Z 48,A -2.4793,B 0,C 0,E1 0.1598,E2 90.072} C_DIS
LIN {X 6.5828,Y -0.7219,Z 48,A -2.4465,B 0,C 0,E1 0.1598,E2 90.072} C_DIS
LIN {X 6.6182,Y -0.0411,Z 48,A -2.4161,B 0,C 0,E1 0.1598,E2 90.072} C_DIS
LIN {X 6.5882,Y 0.6397,Z 48,A -2.3881,B 0,C 0,E1 0.1598,E2 90.0721} C_DIS
LIN {X 6.4872,Y 1.3138,Z 48,A -2.3631,B 0,C 0,E1 0.1598,E2 90.0721} C_DIS
LIN {X 6.3206,Y 1.9748,Z 48,A -2.341,B 0,C 0,E1 0.1598,E2 90.0721} C_DIS
LIN {X 6.0844,Y 2.6142,Z 48,A -2.3225,B 0,C 0,E1 0.1598,E2 90.0722} C_DIS
LIN {X 5.7831,Y 3.2256,Z 48,A -2.3075,B 0,C 0,E1 0.1598,E2 90.0722} C_DIS
LIN {X 5.4206,Y 3.803,Z 48,A -2.2963,B 0,C 0,E1 0.1598,E2 90.0723} C_DIS
LIN {X 4.9998,Y 4.3392,Z 48,A -2.2889,B 0,C 0,E1 0.1598,E2 90.0723} C_DIS
LIN {X 4.5275,Y 4.8309,Z 48,A -2.2854,B 0,C 0,E1 0.1598,E2 90.0723} C_DIS
LIN {X 4.0074,Y 5.2715,Z 48,A -2.2859,B 0,C 0,E1 0.1598,E2 90.0723} C_DIS
LIN {X 3.4429,Y 5.6537,Z 48,A -2.2904,B 0,C 0,E1 0.1598,E2 90.0724} C_DIS
LIN {X 2.8434,Y 5.9781,Z 48,A -2.2988,B 0,C 0,E1 0.1598,E2 90.0724} C_DIS
LIN {X 2.2142,Y 6.2402,Z 48,A -2.3109,B 0,C 0,E1 0.1598,E2 90.0724} C_DIS
LIN {X 1.5607,Y 6.4335,Z 48,A -2.3268,B 0,C 0,E1 0.1598,E2 90.0724} C_DIS
LIN {X 0.8908,Y 6.5597,Z 48,A -2.3461,B 0,C 0,E1 0.1598,E2 90.0724} C_DIS
LIN {X 0.2115,Y 6.615,Z 48,A -2.3689,B 0,C 0,E1 0.1598,E2 90.0724} C_DIS
LIN {X -0.47,Y 6.6049,Z 48,A -2.3944,B 0,C 0,E1 0.1598,E2 90.0724} C_DIS
LIN {X -1.1465,Y 6.5209,Z 48,A -2.423,B 0,C 0,E1 0.1598,E2 90.0724} C_DIS
LIN {X -1.8105,Y 6.3672,Z 48,A -2.454,B 0,C 0,E1 0.1598,E2 90.0723} C_DIS
LIN {X -2.4558,Y 6.1478,Z 48,A -2.4871,B 0,C 0,E1 0.1598,E2 90.0723} C_DIS
LIN {X -3.0747,Y 5.8624,Z 48,A -2.522,B 0,C 0,E1 0.1598,E2 90.0722} C_DIS
LIN {X -3.6612,Y 5.5151,Z 48,A -2.5583,B 0,C 0,E1 0.1598,E2 90.0722} C_DIS
LIN {X -4.2088,Y 5.1094,Z 48,A -2.5957,B 0,C 0,E1 0.1598,E2 90.072} C_DIS
LIN {X -4.7112,Y 4.649,Z 48,A -2.6337,B 0,C 0,E1 0.1598,E2 90.072} C_DIS
LIN {X -5.1644,Y 4.1399,Z 48,A -2.6719,B 0,C 0,E1 0.1598,E2 90.0719} C_DIS
LIN {X -5.5636,Y 3.5874,Z 48,A -2.71,B 0,C 0,E1 0.1598,E2 90.0719} C_DIS
LIN {X -5.9029,Y 2.9963,Z 48,A -2.7475,B 0,C 0,E1 0.1598,E2 90.0717} C_DIS
LIN {X -6.1804,Y 2.3737,Z 48,A -2.784,B 0,C 0,E1 0.1598,E2 90.0717} C_DIS
LIN {X -6.3927,Y 1.7261,Z 48,A -2.8193,B 0,C 0,E1 0.1598,E2 90.0716} C_DIS
LIN {X -6.5371,Y 1.0599,Z 48,A -2.8528,B 0,C 0,E1 0.1598,E2 90.0716} C_DIS
LIN {X -6.6105,Y 0.3821,Z 48,A -2.8842,B 0,C 0,E1 0.1598,E2 90.0715} C_DIS
LIN {X -6.6116,Y -0.2995,Z 48,A -2.9131,B 0,C 0,E1 0.1598,E2 90.0715} C_DIS
LIN {X -6.5489,Y -0.9782,Z 48,A -2.9396,B 0,C 0,E1 0.1598,E2 90.0715} C_DIS
LIN {X -6.4144,Y -1.6465,Z 48,A -2.9629,B 0,C 0,E1 0.1598,E2 90.0714} C_DIS
LIN {X -6.2113,Y -2.2972,Z 48,A -2.9831,B 0,C 0,E1 0.1598,E2 90.0714} C_DIS
LIN {X -5.9418,Y -2.9234,Z 48,A -2.9998,B 0,C 0,E1 0.1598,E2 90.0714} C_DIS
LIN {X -5.6084,Y -3.5178,Z 48,A -3.0127,B 0,C 0,E1 0.1598,E2 90.0714} C_DIS
LIN {X -5.2169,Y -4.076,Z 48,A -3.0221,B 0,C 0,E1 0.1598,E2 90.0714} C_DIS
LIN {X -4.7712,Y -4.5917,Z 48,A -3.0276,B 0,C 0,E1 0.1598,E2 90.0714} C_DIS
LIN {X -4.2726,Y -5.0565,Z 48,A -3.0291,B 0,C 0,E1 0.1598,E2 90.0714} C_DIS
LIN {X -3.7291,Y -5.4679,Z 48,A -3.0267,B 0,C 0,E1 0.1598,E2 90.0714} C_DIS
LIN {X -3.1473,Y -5.8229,Z 48,A -3.0204,B 0,C 0,E1 0.1598,E2 90.0714} C_DIS
LIN {X -2.5326,Y -6.1175,Z 48,A -3.0104,B 0,C 0,E1 0.1598,E2 90.0715} C_DIS
LIN {X -1.8904,Y -6.3456,Z 48,A -2.9966,B 0,C 0,E1 0.1598,E2 90.0715} C_DIS
LIN {X -1.2279,Y -6.5058,Z 48,A -2.9791,B 0,C 0,E1 0.1598,E2 90.0715} C_DIS
LIN {X -0.5526,Y -6.5981,Z 48,A -2.9583,B 0,C 0,E1 0.1598,E2 90.0716} C_DIS
LIN {X -0.5526,Y -6.5981,Z 48,A -2.9583,B 0,C 0,E1 0.1598,E2 90.0716} C_DIS
Enddeposition()
LIN {X -0.0328,Y -7.5551,Z 48,A -2.979,B 0,C 0,E1 0.1598,E2 90.0704} C_DIS
Startdeposition()
$VEL.CP = VEL_PRINT
LIN {X -0.8366,Y -7.5071,Z 48,A -3.0075,B 0,C 0,E1 0.1598,E2 90.0715} C_DIS
LIN {X -1.6319,Y -7.3789,Z 48,A -3.0313,B 0,C 0,E1 0.1598,E2 90.0715} C_DIS
LIN {X -2.8981,Y -6.979,Z 48,A -3.0606,B 0,C 0,E1 0.1598,E2 90.0714} C_DIS
LIN {X -3.8726,Y -6.4897,Z 48,A -3.0755,B 0,C 0,E1 0.1598,E2 90.0714} C_DIS
LIN {X -4.6612,Y -5.9432,Z 48,A -3.0812,B 0,C 0,E1 0.1598,E2 90.0714} C_DIS
LIN {X -5.5097,Y -5.1715,Z 48,A -3.0794,B 0,C 0,E1 0.1598,E2 90.0711} C_DIS
LIN {X -6.1481,Y -4.3949,Z 48,A -3.0698,B 0,C 0,E1 0.1598,E2 90.0711} C_DIS
LIN {X -6.6645,Y -3.5559,Z 48,A -3.0532,B 0,C 0,E1 0.1598,E2 90.0711} C_DIS
LIN {X -6.997,Y -2.8412,Z 48,A -3.0352,B 0,C 0,E1 0.1598,E2 90.0712} C_DIS
LIN {X -7.3119,Y -1.9077,Z 48,A -3.0069,B 0,C 0,E1 0.1598,E2 90.071} C_DIS
LIN {X -7.5229,Y -0.6763,Z 48,A -2.9622,B 0,C 0,E1 0.1598,E2 90.0708} C_DIS
LIN {X -7.5549,Y 0.1745,Z 48,A -2.9276,B 0,C 0,E1 0.1598,E2 90.0711} C_DIS
LIN {X -7.4392,Y 1.3107,Z 48,A -2.8751,B 0,C 0,E1 0.1598,E2 90.0711} C_DIS
LIN {X -7.2716,Y 2.0585,Z 48,A -2.8375,B 0,C 0,E1 0.1598,E2 90.0713} C_DIS
LIN {X -6.8991,Y 3.0828,Z 48,A -2.7803,B 0,C 0,E1 0.1598,E2 90.0713} C_DIS
LIN {X -6.2055,Y 4.3036,Z 48,A -2.7029,B 0,C 0,E1 0.1598,E2 90.0713} C_DIS
LIN {X -5.4976,Y 5.1842,Z 48,A -2.6398,B 0,C 0,E1 0.1598,E2 90.0717} C_DIS
LIN {X -4.7593,Y 5.8717,Z 48,A -2.5836,B 0,C 0,E1 0.1598,E2 90.0718} C_DIS
LIN {X -3.9241,Y 6.4579,Z 48,A -2.5281,B 0,C 0,E1 0.1598,E2 90.072} C_DIS
LIN {X -3.0346,Y 6.921,Z 48,A -2.4757,B 0,C 0,E1 0.1598,E2 90.0722} C_DIS
LIN {X -2.1171,Y 7.2555,Z 48,A -2.4277,B 0,C 0,E1 0.1598,E2 90.0722} C_DIS
LIN {X -0.9574,Y 7.4967,Z 48,A -2.3747,B 0,C 0,E1 0.1598,E2 90.0724} C_DIS
LIN {X 0.0575,Y 7.5576,Z 48,A -2.3347,B 0,C 0,E1 0.1598,E2 90.0724} C_DIS
LIN {X 0.8935,Y 7.504,Z 48,A -2.3061,B 0,C 0,E1 0.1598,E2 90.0724} C_DIS
LIN {X 2.01,Y 7.2812,Z 48,A -2.2743,B 0,C 0,E1 0.1598,E2 90.0724} C_DIS
LIN {X 3.07,Y 6.9059,Z 48,A -2.2511,B 0,C 0,E1 0.1598,E2 90.0724} C_DIS
LIN {X 3.9693,Y 6.4245,Z 48,A -2.2384,B 0,C 0,E1 0.1598,E2 90.0724} C_DIS
LIN {X 4.6393,Y 5.9587,Z 48,A -2.2335,B 0,C 0,E1 0.1598,E2 90.0724} C_DIS
LIN {X 5.2569,Y 5.4253,Z 48,A -2.2335,B 0,C 0,E1 0.1598,E2 90.0724} C_DIS
LIN {X 5.9417,Y 4.6692,Z 48,A -2.2402,B 0,C 0,E1 0.1598,E2 90.0722} C_DIS
LIN {X 6.6141,Y 3.651,Z 48,A -2.2586,B 0,C 0,E1 0.1598,E2 90.0719} C_DIS
LIN {X 6.9579,Y 2.9478,Z 48,A -2.276,B 0,C 0,E1 0.1598,E2 90.0721} C_DIS
LIN {X 7.3215,Y 1.8707,Z 48,A -2.3085,B 0,C 0,E1 0.1598,E2 90.0719} C_DIS
LIN {X 7.5174,Y 0.7219,Z 48,A -2.3501,B 0,C 0,E1 0.1598,E2 90.0716} C_DIS
LIN {X 7.5503,Y -0.1136,Z 48,A -2.3849,B 0,C 0,E1 0.1598,E2 90.072} C_DIS
LIN {X 7.4926,Y -0.9478,Z 48,A -2.4227,B 0,C 0,E1 0.1598,E2 90.072} C_DIS
LIN {X 7.2946,Y -1.9742,Z 48,A -2.4736,B 0,C 0,E1 0.1598,E2 90.0716} C_DIS
LIN {X 6.9251,Y -3.0135,Z 48,A -2.5316,B 0,C 0,E1 0.1598,E2 90.0716} C_DIS
LIN {X 6.4675,Y -3.9086,Z 48,A -2.5867,B 0,C 0,E1 0.1598,E2 90.0716} C_DIS
LIN {X 5.8781,Y -4.7518,Z 48,A -2.6445,B 0,C 0,E1 0.1598,E2 90.0717} C_DIS
LIN {X 5.0871,Y -5.5828,Z 48,A -2.709,B 0,C 0,E1 0.1598,E2 90.0716} C_DIS
LIN {X 4.2052,Y -6.2792,Z 48,A -2.7712,B 0,C 0,E1 0.1598,E2 90.0716} C_DIS
LIN {X 3.2335,Y -6.825,Z 48,A -2.8302,B 0,C 0,E1 0.1598,E2 90.0716} C_DIS
LIN {X 2.5217,Y -7.1205,Z 48,A -2.8691,B 0,C 0,E1 0.1598,E2 90.0717} C_DIS
LIN {X 1.783,Y -7.34,Z 48,A -2.9055,B 0,C 0,E1 0.1598,E2 90.0717} C_DIS
LIN {X 0.7109,Y -7.5247,Z 48,A -2.9527,B 0,C 0,E1 0.1598,E2 90.0717} C_DIS
LIN {X -0.0328,Y -7.5551,Z 48,A -2.9813,B 0,C 0,E1 0.1598,E2 90.0717} C_DIS
Enddeposition()
LIN {X -0.0328,Y -7.5551,Z 48,A -2.9813,B 0,C 0,E1 0.1598,E2 90.0717} C_DIS
Startdeposition()
$VEL.CP = VEL_PRINT
LIN {X 0.5229,Y -8.4709,Z 48,A -2.9995,B 0,C 0,E1 0.1598,E2 90.071} C_DIS
LIN {X 1.2949,Y -8.3864,Z 48,A -2.9682,B 0,C 0,E1 0.1598,E2 90.0716} C_DIS
LIN {X 2.0561,Y -8.2329,Z 48,A -2.9338,B 0,C 0,E1 0.1598,E2 90.0716} C_DIS
LIN {X 2.8005,Y -8.0113,Z 48,A -2.897,B 0,C 0,E1 0.1598,E2 90.0716} C_DIS
LIN {X 3.9381,Y -7.5235,Z 48,A -2.8344,B 0,C 0,E1 0.1598,E2 90.0716} C_DIS
LIN {X 5.0242,Y -6.8401,Z 48,A -2.7653,B 0,C 0,E1 0.1598,E2 90.0716} C_DIS
LIN {X 5.6985,Y -6.2889,Z 48,A -2.7171,B 0,C 0,E1 0.1598,E2 90.0718} C_DIS
LIN {X 6.3128,Y -5.6716,Z 48,A -2.6681,B 0,C 0,E1 0.1598,E2 90.0718} C_DIS
LIN {X 6.8607,Y -4.9946,Z 48,A -2.6191,B 0,C 0,E1 0.1598,E2 90.0718} C_DIS
LIN {X 7.4469,Y -4.0773,Z 48,A -2.5581,B 0,C 0,E1 0.1598,E2 90.0716} C_DIS
LIN {X 7.8296,Y -3.2836,Z 48,A -2.5103,B 0,C 0,E1 0.1598,E2 90.0719} C_DIS
LIN {X 8.1757,Y -2.2955,Z 48,A -2.4551,B 0,C 0,E1 0.1598,E2 90.0718} C_DIS
LIN {X 8.4115,Y -1.1295,Z 48,A -2.3963,B 0,C 0,E1 0.1598,E2 90.0716} C_DIS
LIN {X 8.4845,Y -0.2547,Z 48,A -2.3566,B 0,C 0,E1 0.1598,E2 90.072} C_DIS
LIN {X 8.4656,Y 0.6229,Z 48,A -2.3198,B 0,C 0,E1 0.1598,E2 90.072} C_DIS
LIN {X 8.3551,Y 1.4939,Z 48,A -2.2867,B 0,C 0,E1 0.1598,E2 90.072} C_DIS
LIN {X 8.1554,Y 2.3488,Z 48,A -2.2575,B 0,C 0,E1 0.1598,E2 90.0721} C_DIS
LIN {X 7.8695,Y 3.1789,Z 48,A -2.2326,B 0,C 0,E1 0.1598,E2 90.0721} C_DIS
LIN {X 7.4993,Y 3.9749,Z 48,A -2.2123,B 0,C 0,E1 0.1598,E2 90.0722} C_DIS
LIN {X 6.9264,Y 4.9108,Z 48,A -2.1933,B 0,C 0,E1 0.1598,E2 90.072} C_DIS
LIN {X 6.1364,Y 5.8653,Z 48,A -2.1817,B 0,C 0,E1 0.1598,E2 90.072} C_DIS
LIN {X 5.5433,Y 6.4306,Z 48,A -2.1798,B 0,C 0,E1 0.1598,E2 90.0723} C_DIS
LIN {X 4.6962,Y 7.0692,Z 48,A -2.1839,B 0,C 0,E1 0.1598,E2 90.0724} C_DIS
LIN {X 3.9665,Y 7.5027,Z 48,A -2.1925,B 0,C 0,E1 0.1598,E2 90.0725} C_DIS
LIN {X 3.1973,Y 7.8612,Z 48,A -2.2057,B 0,C 0,E1 0.1598,E2 90.0725} C_DIS
LIN {X 2.3962,Y 8.1411,Z 48,A -2.2234,B 0,C 0,E1 0.1598,E2 90.0725} C_DIS
LIN {X 1.5711,Y 8.3397,Z 48,A -2.2455,B 0,C 0,E1 0.1598,E2 90.0725} C_DIS
LIN {X 0.7304,Y 8.4554,Z 48,A -2.2716,B 0,C 0,E1 0.1598,E2 90.0725} C_DIS
LIN {X -0.1176,Y 8.4866,Z 48,A -2.3016,B 0,C 0,E1 0.1598,E2 90.0725} C_DIS
LIN {X -0.9643,Y 8.431,Z 48,A -2.3352,B 0,C 0,E1 0.1598,E2 90.0725} C_DIS
LIN {X -1.8014,Y 8.2919,Z 48,A -2.372,B 0,C 0,E1 0.1598,E2 90.0724} C_DIS
LIN {X -2.6205,Y 8.0704,Z 48,A -2.4116,B 0,C 0,E1 0.1598,E2 90.0724} C_DIS
LIN {X -3.4134,Y 7.7682,Z 48,A -2.4537,B 0,C 0,E1 0.1598,E2 90.0723} C_DIS
LIN {X -4.5097,Y 7.1935,Z 48,A -2.5184,B 0,C 0,E1 0.1598,E2 90.0721} C_DIS
LIN {X -5.3429,Y 6.5935,Z 48,A -2.5745,B 0,C 0,E1 0.1598,E2 90.072} C_DIS
LIN {X -5.9549,Y 6.0457,Z 48,A -2.6203,B 0,C 0,E1 0.1598,E2 90.072} C_DIS
LIN {X -6.6452,Y 5.2858,Z 48,A -2.6777,B 0,C 0,E1 0.1598,E2 90.0717} C_DIS
LIN {X -7.2955,Y 4.3377,Z 48,A -2.7416,B 0,C 0,E1 0.1598,E2 90.0714} C_DIS
LIN {X -7.8131,Y 3.3224,Z 48,A -2.8036,B 0,C 0,E1 0.1598,E2 90.0714} C_DIS
LIN {X -8.1526,Y 2.357,Z 48,A -2.857,B 0,C 0,E1 0.1598,E2 90.0714} C_DIS
LIN {X -8.3415,Y 1.5604,Z 48,A -2.8978,B 0,C 0,E1 0.1598,E2 90.0714} C_DIS
LIN {X -8.4539,Y 0.7495,Z 48,A -2.9362,B 0,C 0,E1 0.1598,E2 90.0714} C_DIS
LIN {X -8.4872,Y -0.0684,Z 48,A -2.9721,B 0,C 0,E1 0.1598,E2 90.0713} C_DIS
LIN {X -8.3938,Y -1.2793,Z 48,A -3.0195,B 0,C 0,E1 0.1598,E2 90.0708} C_DIS
LIN {X -8.1667,Y -2.3109,Z 48,A -3.055,B 0,C 0,E1 0.1598,E2 90.071} C_DIS
LIN {X -7.8961,Y -3.1115,Z 48,A -3.0792,B 0,C 0,E1 0.1598,E2 90.0711} C_DIS
LIN {X -7.5472,Y -3.881,Z 48,A -3.099,B 0,C 0,E1 0.1598,E2 90.0711} C_DIS
LIN {X -7.1234,Y -4.6121,Z 48,A -3.1145,B 0,C 0,E1 0.1598,E2 90.0711} C_DIS
LIN {X -6.6292,Y -5.2974,Z 48,A -3.1254,B 0,C 0,E1 0.1598,E2 90.0711} C_DIS
LIN {X -5.8535,Y -6.1495,Z 48,A -3.133,B 0,C 0,E1 0.1598,E2 90.0711} C_DIS
LIN {X -5.0545,Y -6.8175,Z 48,A -3.1322,B 0,C 0,E1 0.1598,E2 90.0711} C_DIS
LIN {X -4.3615,Y -7.2799,Z 48,A -3.1266,B 0,C 0,E1 0.1598,E2 90.0713} C_DIS
LIN {X -3.6265,Y -7.6722,Z 48,A -3.1163,B 0,C 0,E1 0.1598,E2 90.0713} C_DIS
LIN {X -2.5507,Y -8.0981,Z 48,A -3.095,B 0,C 0,E1 0.1598,E2 90.0713} C_DIS
LIN {X -1.5905,Y -8.3361,Z 48,A -3.07,B 0,C 0,E1 0.1598,E2 90.0714} C_DIS
LIN {X -0.4425,Y -8.48,Z 48,A -3.0341,B 0,C 0,E1 0.1598,E2 90.0715} C_DIS
LIN {X -0.4425,Y -8.48,Z 48,A -3.0341,B 0,C 0,E1 0.1598,E2 90.0715} C_DIS
Enddeposition()
LIN {X 0.0009,Y -4.7524,Z 49,A -2.8446,B 0,C 0,E1 0.1598,E2 90.0604} C_DIS
Startdeposition()
$VEL.CP = VEL_PRINT
LIN {X 0.0009,Y -4.7524,Z 49,A -2.8503,B 0,C 0,E1 0.1598,E2 90.0661} C_DIS
LIN {X -0.653,Y -4.7048,Z 49,A -2.8772,B 0,C 0,E1 0.1598,E2 90.0711} C_DIS
LIN {X -1.4522,Y -4.5251,Z 49,A -2.8995,B 0,C 0,E1 0.1598,E2 90.0716} C_DIS
LIN {X -2.0612,Y -4.2819,Z 49,A -2.9116,B 0,C 0,E1 0.1598,E2 90.0716} C_DIS
LIN {X -2.6305,Y -3.9568,Z 49,A -2.9186,B 0,C 0,E1 0.1598,E2 90.0716} C_DIS
LIN {X -3.1503,Y -3.5572,Z 49,A -2.9207,B 0,C 0,E1 0.1598,E2 90.0716} C_DIS
LIN {X -3.6095,Y -3.0892,Z 49,A -2.9176,B 0,C 0,E1 0.1598,E2 90.0716} C_DIS
LIN {X -4.0004,Y -2.563,Z 49,A -2.9096,B 0,C 0,E1 0.1598,E2 90.0716} C_DIS
LIN {X -4.3155,Y -1.9881,Z 49,A -2.8968,B 0,C 0,E1 0.1598,E2 90.0716} C_DIS
LIN {X -4.5479,Y -1.375,Z 49,A -2.8792,B 0,C 0,E1 0.1598,E2 90.0716} C_DIS
LIN {X -4.6941,Y -0.736,Z 49,A -2.8575,B 0,C 0,E1 0.1598,E2 90.0716} C_DIS
LIN {X -4.7508,Y -0.0829,Z 49,A -2.8319,B 0,C 0,E1 0.1598,E2 90.0716} C_DIS
LIN {X -4.7163,Y 0.5717,Z 49,A -2.8028,B 0,C 0,E1 0.1598,E2 90.0716} C_DIS
LIN {X -4.5928,Y 1.2155,Z 49,A -2.771,B 0,C 0,E1 0.1598,E2 90.0716} C_DIS
LIN {X -4.3816,Y 1.836,Z 49,A -2.7369,B 0,C 0,E1 0.1598,E2 90.0717} C_DIS
LIN {X -4.0869,Y 2.4215,Z 49,A -2.7012,B 0,C 0,E1 0.1598,E2 90.0717} C_DIS
LIN {X -3.7151,Y 2.9613,Z 49,A -2.6647,B 0,C 0,E1 0.1598,E2 90.0719} C_DIS
LIN {X -3.2716,Y 3.4441,Z 49,A -2.6279,B 0,C 0,E1 0.1598,E2 90.0719} C_DIS
LIN {X -2.7666,Y 3.862,Z 49,A -2.5916,B 0,C 0,E1 0.1598,E2 90.072} C_DIS
LIN {X -2.2087,Y 4.2063,Z 49,A -2.5564,B 0,C 0,E1 0.1598,E2 90.0721} C_DIS
LIN {X -1.6086,Y 4.4699,Z 49,A -2.5232,B 0,C 0,E1 0.1598,E2 90.0721} C_DIS
LIN {X -0.9782,Y 4.6497,Z 49,A -2.4923,B 0,C 0,E1 0.1598,E2 90.0722} C_DIS
LIN {X -0.3286,Y 4.7386,Z 49,A -2.4646,B 0,C 0,E1 0.1598,E2 90.0722} C_DIS
LIN {X 0.3268,Y 4.7396,Z 49,A -2.4404,B 0,C 0,E1 0.1598,E2 90.0723} C_DIS
LIN {X 0.976,Y 4.6495,Z 49,A -2.4203,B 0,C 0,E1 0.1598,E2 90.0723} C_DIS
LIN {X 1.6067,Y 4.4708,Z 49,A -2.4046,B 0,C 0,E1 0.1598,E2 90.0723} C_DIS
LIN {X 2.2071,Y 4.2076,Z 49,A -2.3937,B 0,C 0,E1 0.1598,E2 90.0723} C_DIS
LIN {X 2.765,Y 3.8633,Z 49,A -2.3878,B 0,C 0,E1 0.1598,E2 90.0723} C_DIS
LIN {X 3.2703,Y 3.4457,Z 49,A -2.3869,B 0,C 0,E1 0.1598,E2 90.0723} C_DIS
LIN {X 3.7139,Y 2.9631,Z 49,A -2.3911,B 0,C 0,E1 0.1598,E2 90.0723} C_DIS
LIN {X 4.0865,Y 2.4236,Z 49,A -2.4003,B 0,C 0,E1 0.1598,E2 90.0722} C_DIS
LIN {X 4.3817,Y 1.8383,Z 49,A -2.4143,B 0,C 0,E1 0.1598,E2 90.0722} C_DIS
LIN {X 4.593,Y 1.2176,Z 49,A -2.433,B 0,C 0,E1 0.1598,E2 90.0722} C_DIS
LIN {X 4.7157,Y 0.5737,Z 49,A -2.4559,B 0,C 0,E1 0.1598,E2 90.0721} C_DIS
LIN {X 4.7509,Y -0.0809,Z 49,A -2.4825,B 0,C 0,E1 0.1598,E2 90.0721} C_DIS
LIN {X 4.6956,Y -0.7343,Z 49,A -2.5124,B 0,C 0,E1 0.1598,E2 90.072} C_DIS
LIN {X 4.55,Y -1.3737,Z 49,A -2.5451,B 0,C 0,E1 0.1598,E2 90.072} C_DIS
LIN {X 4.3164,Y -1.9863,Z 49,A -2.5798,B 0,C 0,E1 0.1598,E2 90.072} C_DIS
LIN {X 4.0012,Y -2.5611,Z 49,A -2.6159,B 0,C 0,E1 0.1598,E2 90.072} C_DIS
LIN {X 3.6117,Y -3.0886,Z 49,A -2.6527,B 0,C 0,E1 0.1598,E2 90.0719} C_DIS
LIN {X 3.1525,Y -3.5568,Z 49,A -2.6896,B 0,C 0,E1 0.1598,E2 90.0719} C_DIS
LIN {X 2.6318,Y -3.9553,Z 49,A -2.7258,B 0,C 0,E1 0.1598,E2 90.0719} C_DIS
LIN {X 2.0624,Y -4.2801,Z 49,A -2.7605,B 0,C 0,E1 0.1598,E2 90.0719} C_DIS
LIN {X 1.4536,Y -4.5237,Z 49,A -2.7933,B 0,C 0,E1 0.1598,E2 90.0719} C_DIS
LIN {X 0.8173,Y -4.6826,Z 49,A -2.8234,B 0,C 0,E1 0.1598,E2 90.0719} C_DIS
LIN {X 0.0009,Y -4.7524,Z 49,A -2.8564,B 0,C 0,E1 0.1598,E2 90.0718} C_DIS
Enddeposition()
LIN {X 0.0009,Y -4.7524,Z 49,A -2.8564,B 0,C 0,E1 0.1598,E2 90.0718} C_DIS
Startdeposition()
$VEL.CP = VEL_PRINT
LIN {X 0.5093,Y -5.6629,Z 49,A -2.876,B 0,C 0,E1 0.1598,E2 90.0711} C_DIS
LIN {X 1.2145,Y -5.5554,Z 49,A -2.8461,B 0,C 0,E1 0.1598,E2 90.0717} C_DIS
LIN {X 1.8999,Y -5.3578,Z 49,A -2.8126,B 0,C 0,E1 0.1598,E2 90.0718} C_DIS
LIN {X 2.5556,Y -5.077,Z 49,A -2.7765,B 0,C 0,E1 0.1598,E2 90.0718} C_DIS
LIN {X 3.1713,Y -4.7169,Z 49,A -2.7385,B 0,C 0,E1 0.1598,E2 90.0718} C_DIS
LIN {X 3.7381,Y -4.2837,Z 49,A -2.6992,B 0,C 0,E1 0.1598,E2 90.0718} C_DIS
LIN {X 4.2452,Y -3.7817,Z 49,A -2.6591,B 0,C 0,E1 0.1598,E2 90.0718} C_DIS
LIN {X 4.6834,Y -3.2188,Z 49,A -2.619,B 0,C 0,E1 0.1598,E2 90.0719} C_DIS
LIN {X 5.0517,Y -2.608,Z 49,A -2.5794,B 0,C 0,E1 0.1598,E2 90.0719} C_DIS
LIN {X 5.449,Y -1.6377,Z 49,A -2.523,B 0,C 0,E1 0.1598,E2 90.0717} C_DIS
LIN {X 5.6467,Y -0.6396,Z 49,A -2.4732,B 0,C 0,E1 0.1598,E2 90.0717} C_DIS
LIN {X 5.6813,Y 0.1737,Z 49,A -2.4373,B 0,C 0,E1 0.1598,E2 90.0719} C_DIS
LIN {X 5.6003,Y 0.9839,Z 49,A -2.4057,B 0,C 0,E1 0.1598,E2 90.0719} C_DIS
LIN {X 5.3991,Y 1.7729,Z 49,A -2.3795,B 0,C 0,E1 0.1598,E2 90.072} C_DIS
LIN {X 5.0909,Y 2.5263,Z 49,A -2.3587,B 0,C 0,E1 0.1598,E2 90.072} C_DIS
LIN {X 4.6787,Y 3.2282,Z 49,A -2.344,B 0,C 0,E1 0.1598,E2 90.0721} C_DIS
LIN {X 4.1687,Y 3.8628,Z 49,A -2.3358,B 0,C 0,E1 0.1598,E2 90.0722} C_DIS
LIN {X 3.5738,Y 4.4184,Z 49,A -2.3342,B 0,C 0,E1 0.1598,E2 90.0722} C_DIS
LIN {X 2.9062,Y 4.884,Z 49,A -2.339,B 0,C 0,E1 0.1598,E2 90.0723} C_DIS
LIN {X 2.178,Y 5.2475,Z 49,A -2.3504,B 0,C 0,E1 0.1598,E2 90.0723} C_DIS
LIN {X 1.4061,Y 5.5053,Z 49,A -2.368,B 0,C 0,E1 0.1598,E2 90.0723} C_DIS
LIN {X 0.6053,Y 5.651,Z 49,A -2.3913,B 0,C 0,E1 0.1598,E2 90.0723} C_DIS
LIN {X -0.5769,Y 5.6607,Z 49,A -2.4345,B 0,C 0,E1 0.1598,E2 90.0723} C_DIS
LIN {X -1.5497,Y 5.4751,Z 49,A -2.4783,B 0,C 0,E1 0.1598,E2 90.0723} C_DIS
LIN {X -2.6853,Y 5.016,Z 49,A -2.5395,B 0,C 0,E1 0.1598,E2 90.0721} C_DIS
LIN {X -3.4646,Y 4.5084,Z 49,A -2.5898,B 0,C 0,E1 0.1598,E2 90.0721} C_DIS
LIN {X -4.0782,Y 3.9591,Z 49,A -2.6356,B 0,C 0,E1 0.1598,E2 90.0719} C_DIS
LIN {X -4.6059,Y 3.3272,Z 49,A -2.6818,B 0,C 0,E1 0.1598,E2 90.0718} C_DIS
LIN {X -5.0402,Y 2.6278,Z 49,A -2.7274,B 0,C 0,E1 0.1598,E2 90.0717} C_DIS
LIN {X -5.4365,Y 1.6777,Z 49,A -2.782,B 0,C 0,E1 0.1598,E2 90.0713} C_DIS
LIN {X -5.6865,Y 0.2102,Z 49,A -2.8528,B 0,C 0,E1 0.1598,E2 90.0706} C_DIS
LIN {X -5.6288,Y -0.7778,Z 49,A -2.8932,B 0,C 0,E1 0.1598,E2 90.0712} C_DIS
LIN {X -5.4671,Y -1.5528,Z 49,A -2.9202,B 0,C 0,E1 0.1598,E2 90.0713} C_DIS
LIN {X -5.1982,Y -2.2974,Z 49,A -2.942,B 0,C 0,E1 0.1598,E2 90.0713} C_DIS
LIN {X -4.8294,Y -2.998,Z 49,A -2.9582,B 0,C 0,E1 0.1598,E2 90.0713} C_DIS
LIN {X -4.3658,Y -3.6399,Z 49,A -2.9685,B 0,C 0,E1 0.1598,E2 90.0713} C_DIS
LIN {X -3.8181,Y -4.2118,Z 49,A -2.9727,B 0,C 0,E1 0.1598,E2 90.0714} C_DIS
LIN {X -3.1959,Y -4.7019,Z 49,A -2.9707,B 0,C 0,E1 0.1598,E2 90.0714} C_DIS
LIN {X -2.5106,Y -5.0983,Z 49,A -2.9625,B 0,C 0,E1 0.1598,E2 90.0715} C_DIS
LIN {X -1.7778,Y -5.3977,Z 49,A -2.9484,B 0,C 0,E1 0.1598,E2 90.0715} C_DIS
LIN {X -1.0108,Y -5.5951,Z 49,A -2.9287,B 0,C 0,E1 0.1598,E2 90.0716} C_DIS
LIN {X -0.0255,Y -5.6889,Z 49,A -2.8965,B 0,C 0,E1 0.1598,E2 90.0717} C_DIS
Enddeposition()
LIN {X -0.0255,Y -5.6889,Z 49,A -2.8965,B 0,C 0,E1 0.1598,E2 90.0717} C_DIS
Startdeposition()
$VEL.CP = VEL_PRINT
LIN {X -0.5517,Y -6.5982,Z 49,A -2.9541,B 0,C 0,E1 0.1598,E2 90.0711} C_DIS
LIN {X -1.227,Y -6.5059,Z 49,A -2.9755,B 0,C 0,E1 0.1598,E2 90.0716} C_DIS
LIN {X -1.8896,Y -6.3459,Z 49,A -2.993,B 0,C 0,E1 0.1598,E2 90.0716} C_DIS
LIN {X -2.5318,Y -6.1178,Z 49,A -3.0068,B 0,C 0,E1 0.1598,E2 90.0716} C_DIS
LIN {X -3.1466,Y -5.8233,Z 49,A -3.0169,B 0,C 0,E1 0.1598,E2 90.0716} C_DIS
LIN {X -3.7284,Y -5.4684,Z 49,A -3.0231,B 0,C 0,E1 0.1598,E2 90.0715} C_DIS
LIN {X -4.2719,Y -5.0569,Z 49,A -3.0255,B 0,C 0,E1 0.1598,E2 90.0715} C_DIS
LIN {X -4.7706,Y -4.5923,Z 49,A -3.0241,B 0,C 0,E1 0.1598,E2 90.0715} C_DIS
LIN {X -5.2164,Y -4.0766,Z 49,A -3.0185,B 0,C 0,E1 0.1598,E2 90.0715} C_DIS
LIN {X -5.6079,Y -3.5185,Z 49,A -3.0092,B 0,C 0,E1 0.1598,E2 90.0714} C_DIS
LIN {X -5.9414,Y -2.9241,Z 49,A -2.9962,B 0,C 0,E1 0.1598,E2 90.0714} C_DIS
LIN {X -6.211,Y -2.2979,Z 49,A -2.9795,B 0,C 0,E1 0.1598,E2 90.0714} C_DIS
LIN {X -6.4142,Y -1.6472,Z 49,A -2.9593,B 0,C 0,E1 0.1598,E2 90.0714} C_DIS
LIN {X -6.548,Y -0.9789,Z 49,A -2.9359,B 0,C 0,E1 0.1598,E2 90.0714} C_DIS
LIN {X -6.6129,Y -0.3003,Z 49,A -2.9095,B 0,C 0,E1 0.1598,E2 90.0714} C_DIS
LIN {X -6.6107,Y 0.3813,Z 49,A -2.8806,B 0,C 0,E1 0.1598,E2 90.0714} C_DIS
LIN {X -6.5372,Y 1.059,Z 49,A -2.8491,B 0,C 0,E1 0.1598,E2 90.0715} C_DIS
LIN {X -6.3929,Y 1.7252,Z 49,A -2.8156,B 0,C 0,E1 0.1598,E2 90.0715} C_DIS
LIN {X -6.1808,Y 2.373,Z 49,A -2.7804,B 0,C 0,E1 0.1598,E2 90.0716} C_DIS
LIN {X -5.9034,Y 2.9956,Z 49,A -2.7438,B 0,C 0,E1 0.1598,E2 90.0717} C_DIS
LIN {X -5.564,Y 3.5867,Z 49,A -2.7063,B 0,C 0,E1 0.1598,E2 90.0717} C_DIS
LIN {X -5.1649,Y 4.1393,Z 49,A -2.6682,B 0,C 0,E1 0.1598,E2 90.0719} C_DIS
LIN {X -4.7119,Y 4.6484,Z 49,A -2.6299,B 0,C 0,E1 0.1598,E2 90.0719} C_DIS
LIN {X -4.2095,Y 5.109,Z 49,A -2.5919,B 0,C 0,E1 0.1598,E2 90.072} C_DIS
LIN {X -3.662,Y 5.5147,Z 49,A -2.5546,B 0,C 0,E1 0.1598,E2 90.072} C_DIS
LIN {X -3.0756,Y 5.8621,Z 49,A -2.5182,B 0,C 0,E1 0.1598,E2 90.0722} C_DIS
LIN {X -2.4567,Y 6.1475,Z 49,A -2.4833,B 0,C 0,E1 0.1598,E2 90.0722} C_DIS
LIN {X -1.8113,Y 6.367,Z 49,A -2.4502,B 0,C 0,E1 0.1598,E2 90.0722} C_DIS
LIN {X -1.1473,Y 6.5208,Z 49,A -2.4192,B 0,C 0,E1 0.1598,E2 90.0723} C_DIS
LIN {X -0.4709,Y 6.6048,Z 49,A -2.3907,B 0,C 0,E1 0.1598,E2 90.0723} C_DIS
LIN {X 0.2106,Y 6.615,Z 49,A -2.3651,B 0,C 0,E1 0.1598,E2 90.0724} C_DIS
LIN {X 0.8899,Y 6.5599,Z 49,A -2.3424,B 0,C 0,E1 0.1598,E2 90.0724} C_DIS
LIN {X 1.5598,Y 6.4337,Z 49,A -2.323,B 0,C 0,E1 0.1598,E2 90.0724} C_DIS
LIN {X 2.2134,Y 6.2405,Z 49,A -2.3071,B 0,C 0,E1 0.1598,E2 90.0724} C_DIS
LIN {X 2.8426,Y 5.9784,Z 49,A -2.2951,B 0,C 0,E1 0.1598,E2 90.0724} C_DIS
LIN {X 3.4421,Y 5.6542,Z 49,A -2.2867,B 0,C 0,E1 0.1598,E2 90.0724} C_DIS
LIN {X 4.0067,Y 5.272,Z 49,A -2.2821,B 0,C 0,E1 0.1598,E2 90.0724} C_DIS
LIN {X 4.527,Y 4.8315,Z 49,A -2.2817,B 0,C 0,E1 0.1598,E2 90.0724} C_DIS
LIN {X 4.9991,Y 4.3398,Z 49,A -2.2852,B 0,C 0,E1 0.1598,E2 90.0724} C_DIS
LIN {X 5.4201,Y 3.8037,Z 49,A -2.2925,B 0,C 0,E1 0.1598,E2 90.0724} C_DIS
LIN {X 5.7827,Y 3.2264,Z 49,A -2.3037,B 0,C 0,E1 0.1598,E2 90.0723} C_DIS
LIN {X 6.084,Y 2.6149,Z 49,A -2.3187,B 0,C 0,E1 0.1598,E2 90.0723} C_DIS
LIN {X 6.3204,Y 1.9756,Z 49,A -2.3373,B 0,C 0,E1 0.1598,E2 90.0723} C_DIS
LIN {X 6.4864,Y 1.3145,Z 49,A -2.3593,B 0,C 0,E1 0.1598,E2 90.0722} C_DIS
LIN {X 6.5888,Y 0.6406,Z 49,A -2.3843,B 0,C 0,E1 0.1598,E2 90.0722} C_DIS
LIN {X 6.6178,Y -0.0403,Z 49,A -2.4123,B 0,C 0,E1 0.1598,E2 90.0721} C_DIS
LIN {X 6.5828,Y -0.7211,Z 49,A -2.4427,B 0,C 0,E1 0.1598,E2 90.0721} C_DIS
LIN {X 6.47,Y -1.3933,Z 49,A -2.4755,B 0,C 0,E1 0.1598,E2 90.0721} C_DIS
LIN {X 6.2931,Y -2.0515,Z 49,A -2.5101,B 0,C 0,E1 0.1598,E2 90.072} C_DIS
LIN {X 6.0484,Y -2.6876,Z 49,A -2.5463,B 0,C 0,E1 0.1598,E2 90.072} C_DIS
LIN {X 5.7411,Y -3.2959,Z 49,A -2.5836,B 0,C 0,E1 0.1598,E2 90.072} C_DIS
LIN {X 5.3717,Y -3.8686,Z 49,A -2.6216,B 0,C 0,E1 0.1598,E2 90.072} C_DIS
LIN {X 4.946,Y -4.4008,Z 49,A -2.66,B 0,C 0,E1 0.1598,E2 90.0719} C_DIS
LIN {X 4.4669,Y -4.8856,Z 49,A -2.6983,B 0,C 0,E1 0.1598,E2 90.0719} C_DIS
LIN {X 3.9409,Y -5.3193,Z 49,A -2.7362,B 0,C 0,E1 0.1598,E2 90.0719} C_DIS
LIN {X 3.3725,Y -5.6956,Z 49,A -2.7731,B 0,C 0,E1 0.1598,E2 90.0719} C_DIS
LIN {X 2.769,Y -6.0124,Z 49,A -2.8088,B 0,C 0,E1 0.1598,E2 90.0718} C_DIS
LIN {X 2.1361,Y -6.2654,Z 49,A -2.8428,B 0,C 0,E1 0.1598,E2 90.0718} C_DIS
LIN {X 1.4809,Y -6.453,Z 49,A -2.8748,B 0,C 0,E1 0.1598,E2 90.0718} C_DIS
LIN {X 0.8094,Y -6.5705,Z 49,A -2.9045,B 0,C 0,E1 0.1598,E2 90.0717} C_DIS
LIN {X -0.0409,Y -6.6226,Z 49,A -2.9379,B 0,C 0,E1 0.1598,E2 90.0717} C_DIS
Enddeposition()
LIN {X -0.0409,Y -6.6226,Z 49,A -2.9379,B 0,C 0,E1 0.1598,E2 90.0717} C_DIS
Startdeposition()
$VEL.CP = VEL_PRINT
LIN {X 0.5292,Y -7.5373,Z 49,A -2.9555,B 0,C 0,E1 0.1598,E2 90.0711} C_DIS
LIN {X 1.2146,Y -7.4586,Z 49,A -2.9276,B 0,C 0,E1 0.1598,E2 90.0716} C_DIS
LIN {X 2.1539,Y -7.2407,Z 49,A -2.8839,B 0,C 0,E1 0.1598,E2 90.0717} C_DIS
LIN {X 2.8806,Y -6.982,Z 49,A -2.8462,B 0,C 0,E1 0.1598,E2 90.0717} C_DIS
LIN {X 3.7488,Y -6.5622,Z 49,A -2.7964,B 0,C 0,E1 0.1598,E2 90.0717} C_DIS
LIN {X 4.6262,Y -5.9748,Z 49,A -2.7391,B 0,C 0,E1 0.1598,E2 90.0717} C_DIS
LIN {X 5.5241,Y -5.1563,Z 49,A -2.671,B 0,C 0,E1 0.1598,E2 90.0717} C_DIS
LIN {X 6.086,Y -4.4818,Z 49,A -2.6217,B 0,C 0,E1 0.1598,E2 90.0719} C_DIS
LIN {X 6.7571,Y -3.374,Z 49,A -2.5493,B 0,C 0,E1 0.1598,E2 90.0715} C_DIS
LIN {X 7.1507,Y -2.4489,Z 49,A -2.4953,B 0,C 0,E1 0.1598,E2 90.0717} C_DIS
LIN {X 7.42,Y -1.4188,Z 49,A -2.4414,B 0,C 0,E1 0.1598,E2 90.0717} C_DIS
LIN {X 7.5244,Y -0.673,Z 49,A -2.406,B 0,C 0,E1 0.1598,E2 90.072} C_DIS
LIN {X 7.5466,Y 0.4075,Z 49,A -2.3587,B 0,C 0,E1 0.1598,E2 90.0718} C_DIS
LIN {X 7.4386,Y 1.3389,Z 49,A -2.323,B 0,C 0,E1 0.1598,E2 90.072} C_DIS
LIN {X 7.2022,Y 2.2873,Z 49,A -2.2912,B 0,C 0,E1 0.1598,E2 90.072} C_DIS
LIN {X 6.7119,Y 3.475,Z 49,A -2.2583,B 0,C 0,E1 0.1598,E2 90.0718} C_DIS
LIN {X 6.2946,Y 4.1829,Z 49,A -2.244,B 0,C 0,E1 0.1598,E2 90.0723} C_DIS
LIN {X 5.5388,Y 5.1362,Z 49,A -2.2309,B 0,C 0,E1 0.1598,E2 90.0721} C_DIS
LIN {X 4.9522,Y 5.703,Z 49,A -2.2287,B 0,C 0,E1 0.1598,E2 90.0724} C_DIS
LIN {X 4.3075,Y 6.2033,Z 49,A -2.2313,B 0,C 0,E1 0.1598,E2 90.0724} C_DIS
LIN {X 3.6132,Y 6.6318,Z 49,A -2.2387,B 0,C 0,E1 0.1598,E2 90.0724} C_DIS
LIN {X 2.5759,Y 7.1041,Z 49,A -2.2568,B 0,C 0,E1 0.1598,E2 90.0724} C_DIS
LIN {X 1.4325,Y 7.4207,Z 49,A -2.2856,B 0,C 0,E1 0.1598,E2 90.0724} C_DIS
LIN {X 0.3595,Y 7.5498,Z 49,A -2.3198,B 0,C 0,E1 0.1598,E2 90.0724} C_DIS
LIN {X -0.4977,Y 7.5405,Z 49,A -2.3519,B 0,C 0,E1 0.1598,E2 90.0724} C_DIS
LIN {X -1.6191,Y 7.3816,Z 49,A -2.4,B 0,C 0,E1 0.1598,E2 90.0724} C_DIS
LIN {X -2.4803,Y 7.1385,Z 49,A -2.4421,B 0,C 0,E1 0.1598,E2 90.0723} C_DIS
LIN {X -3.4239,Y 6.7377,Z 49,A -2.4938,B 0,C 0,E1 0.1598,E2 90.0722} C_DIS
Enddeposition()
END
